LIN {X 0,Y 193.255,Z 819.241,A -85,B 0,C 180,E1 -22296.988,E2 -22296.988} C_VEL
LIN {X 0,Y 197.064,Z 813.143,A -85,B 0,C 180,E1 -22300.279,E2 -22300.279} C_VEL
LIN {X 0,Y 201.414,Z 805.399,A -85,B 0,C 180,E1 -22303.403,E2 -22303.403} C_VEL
LIN {X 0,Y 205.369,Z 797.537,A -85,B 0,C 180,E1 -22305.868,E2 -22305.868} C_VEL
LIN {X 0,Y 209.515,Z 788.24,A -85,B 0,C 180,E1 -22308.163,E2 -22308.163} C_VEL
LIN {X 0,Y 213.305,Z 778.652,A -85,B 0,C 180,E1 -22310.013,E2 -22310.013} C_VEL
LIN {X 0,Y 216.814,Z 768.226,A -85,B 0,C 180,E1 -22311.613,E2 -22311.613} C_VEL
LIN {X 0,Y 219.996,Z 756.796,A -85,B 0,C 180,E1 -22312.978,E2 -22312.978} C_VEL
LIN {X 0,Y 222.629,Z 744.096,A -85,B 0,C 180,E1 -22314.141,E2 -22314.141} C_VEL
LIN {X 0,Y 224.529,Z 731.563,A -85,B 0,C 180,E1 -22314.927,E2 -22314.927} C_VEL
LIN {X 0,Y 227.202,Z 703.845,A -85,B 0,C 180,E1 -22315.948,E2 -22315.948} C_VEL
LIN {X 0,Y 228.654,Z 686.695,A -85,B 0,C 180,E1 -22316.58,E2 -22316.58} C_VEL
LIN {X 0,Y 224.169,Z 676.859,A -85,B 0,C 180,E1 -22318.997,E2 -22318.997} C_VEL
LIN {X 0,Y 221.19,Z 671.533,A -85,B 0,C 180,E1 -22320.701,E2 -22320.701} C_VEL
LIN {X 0,Y 216.957,Z 664.335,A -85,B 0,C 180,E1 -22323.435,E2 -22323.435} C_VEL
LIN {X 0,Y 214.368,Z 660.748,A -85,B 0,C 180,E1 -22325.332,E2 -22325.332} C_VEL
LIN {X 0,Y 211.647,Z 657.239,A -85,B 0,C 180,E1 -22327.574,E2 -22327.574} C_VEL
LIN {X 0,Y 210.827,Z 655.899,A -85,B 0,C 180,E1 -22328.388,E2 -22328.388} C_VEL
LIN {X 0,Y 208.392,Z 652.958,A -85,B 0,C 180,E1 -22330.962,E2 -22330.962} C_VEL
LIN {X 0,Y 207.628,Z 651.927,A -85,B 0,C 180,E1 -22331.967,E2 -22331.967} C_VEL
LIN {X 0,Y 204.394,Z 648.519,A -85,B 0,C 180,E1 -22338.028,E2 -22338.028} C_VEL
LIN {X 0,Y 203.914,Z 648.189,A -85,B 0,C 180,E1 -22340.162,E2 -22340.162} C_VEL
LIN {X 0,Y 203.877,Z 648.812,A -85,B 0,C 180,E1 -22344.436,E2 -22344.436} C_VEL
LIN {X 0,Y 204.528,Z 650.008,A -85,B 0,C 180,E1 -22347.139,E2 -22347.139} C_VEL
LIN {X 0,Y 206.714,Z 654.204,A -85,B 0,C 180,E1 -22351.648,E2 -22351.648} C_VEL
LIN {X 0,Y 209.182,Z 657.668,A -85,B 0,C 180,E1 -22354.733,E2 -22354.733} C_VEL
LIN {X 0,Y 212.852,Z 664.058,A -85,B 0,C 180,E1 -22358.308,E2 -22358.308} C_VEL
LIN {X 0,Y 216.137,Z 670.151,A -85,B 0,C 180,E1 -22360.912,E2 -22360.912} C_VEL
LIN {X 0,Y 219.121,Z 675.87,A -85,B 0,C 180,E1 -22362.932,E2 -22362.932} C_VEL
LIN {X 0,Y 222.15,Z 682.225,A -85,B 0,C 180,E1 -22364.816,E2 -22364.816} C_VEL
LIN {X 0,Y 225.466,Z 690.402,A -85,B 0,C 180,E1 -22366.748,E2 -22366.748} C_VEL
LIN {X 0,Y 227.388,Z 695.915,A -85,B 0,C 180,E1 -22367.832,E2 -22367.832} C_VEL
LIN {X 0,Y 227.649,Z 702.504,A -85,B 0,C 180,E1 -22368.353,E2 -22368.353} C_VEL
LIN {X 0,Y 226.563,Z 715.23,A -85,B 0,C 180,E1 -22368.815,E2 -22368.815} C_VEL
LIN {X 0,Y 225.654,Z 721.062,A -85,B 0,C 180,E1 -22368.881,E2 -22368.881} C_VEL
LIN {X 0,Y 220.375,Z 740.084,A -85,B 0,C 180,E1 -22368.379,E2 -22368.379} C_VEL
LIN {X 0,Y 219.234,Z 745.859,A -85,B 0,C 180,E1 -22368.517,E2 -22368.517} C_VEL
LIN {X 0,Y 216.729,Z 758.978,A -85,B 0,C 180,E1 -22369.31,E2 -22369.31} C_VEL
LIN {X 0,Y 213.46,Z 771.436,A -85,B 0,C 180,E1 -22370.365,E2 -22370.365} C_VEL
LIN {X 0,Y 209.794,Z 782.932,A -85,B 0,C 180,E1 -22371.704,E2 -22371.704} C_VEL
LIN {X 0,Y 205.342,Z 794.569,A -85,B 0,C 180,E1 -22373.512,E2 -22373.512} C_VEL
LIN {X 0,Y 201.089,Z 804.071,A -85,B 0,C 180,E1 -22375.395,E2 -22375.395} C_VEL
LIN {X 0,Y 196.832,Z 812.801,A -85,B 0,C 180,E1 -22377.617,E2 -22377.617} C_VEL
LIN {X 0,Y 192.143,Z 821.48,A -85,B 0,C 180,E1 -22380.411,E2 -22380.411} C_VEL
LIN {X 0,Y 188.053,Z 828.489,A -85,B 0,C 180,E1 -22383.355,E2 -22383.355} C_VEL
LIN {X 0,Y 184.661,Z 834.168,A -85,B 0,C 180,E1 -22386.446,E2 -22386.446} C_VEL
LIN {X 0,Y 181.753,Z 838.705,A -85,B 0,C 180,E1 -22389.635,E2 -22389.635} C_VEL
LIN {X 0,Y 178.675,Z 843.171,A -85,B 0,C 180,E1 -22394.018,E2 -22394.018} C_VEL
LIN {X 0,Y 177.676,Z 844.782,A -85,B 0,C 180,E1 -22396.271,E2 -22396.271} C_VEL
LIN {X 0,Y 176.453,Z 846.754,A -85,B 0,C 180,E1 -22400.833,E2 -22400.833} C_VEL
LIN {X 0,Y 176.148,Z 847.203,A -85,B 0,C 180,E1 -22405.423,E2 -22405.423} C_VEL
LIN {X 0,Y 176.258,Z 846.809,A -85,B 0,C 180,E1 -22407.715,E2 -22407.715} C_VEL
LIN {X 0,Y 176.431,Z 845.994,A -85,B 0,C 180,E1 -22410,E2 -22410} C_VEL
LIN {X 0,Y 176.296,Z 844.734,A -85,B 0,C 180,E1 -22412.285,E2 -22412.285} C_VEL
LIN {X 0,Y 176.257,Z 841.979,A -85,B 0,C 180,E1 -22415.721,E2 -22415.721} C_VEL
LIN {X 0,Y 176.569,Z 838.131,A -85,B 0,C 180,E1 -22419.161,E2 -22419.161} C_VEL
LIN {X 0,Y 177.28,Z 833.082,A -85,B 0,C 180,E1 -22422.594,E2 -22422.594} C_VEL
LIN {X 0,Y 178.531,Z 826.688,A -85,B 0,C 180,E1 -22425.995,E2 -22425.995} C_VEL
LIN {X 0,Y 180.337,Z 818.624,A -85,B 0,C 180,E1 -22429.345,E2 -22429.345} C_VEL
LIN {X 0,Y 182.337,Z 809.868,A -85,B 0,C 180,E1 -22432.239,E2 -22432.239} C_VEL
LIN {X 0,Y 184.548,Z 800.323,A -85,B 0,C 180,E1 -22434.765,E2 -22434.765} C_VEL
LIN {X 0,Y 186.774,Z 790.459,A -85,B 0,C 180,E1 -22436.842,E2 -22436.842} C_VEL
LIN {X 0,Y 189.283,Z 778.076,A -85,B 0,C 180,E1 -22438.86,E2 -22438.86} C_VEL
LIN {X 0,Y 191.275,Z 766.071,A -85,B 0,C 180,E1 -22440.345,E2 -22440.345} C_VEL
LIN {X 0,Y 192.959,Z 753.018,A -85,B 0,C 180,E1 -22441.495,E2 -22441.495} C_VEL
LIN {X 0,Y 194.105,Z 739.399,A -85,B 0,C 180,E1 -22442.279,E2 -22442.279} C_VEL
LIN {X 0,Y 196.335,Z 697.108,A -85,B 0,C 180,E1 -22444.02,E2 -22444.02} C_VEL
LIN {X 0,Y 193.323,Z 669.983,A -85,B 0,C 180,E1 -22445.752,E2 -22445.752} C_VEL
LIN {X 0,Y 184.7,Z 646.505,A -85,B 0,C 180,E1 -22448.296,E2 -22448.296} C_VEL
LIN {X 0,Y 180.166,Z 635.4,A -85,B 0,C 180,E1 -22449.717,E2 -22449.717} C_VEL
LIN {X 0,Y 178.504,Z 628.254,A -85,B 0,C 180,E1 -22453.774,E2 -22453.774} C_VEL
LIN {X 0,Y 178.451,Z 628.257,A -85,B 0,C 180,E1 -22458.44,E2 -22458.44} C_VEL
LIN {X 0,Y 178.489,Z 628.251,A -85,B 0,C 180,E1 -22461.951,E2 -22461.951} C_VEL
LIN {X 0,Y 178.49,Z 628.253,A -85,B 0,C 180,E1 -22466.546,E2 -22466.546} C_VEL
LIN {X 0,Y 178.522,Z 628.245,A -85,B 0,C 180,E1 -22470.005,E2 -22470.005} C_VEL
LIN {X 0,Y 178.518,Z 628.242,A -85,B 0,C 180,E1 -22474.884,E2 -22474.884} C_VEL
LIN {X 0,Y 178.619,Z 628.229,A -85,B 0,C 180,E1 -22480.785,E2 -22480.785} C_VEL
LIN {X 0,Y 178.657,Z 628.231,A -85,B 0,C 180,E1 -22486.347,E2 -22486.347} C_VEL
LIN {X 0,Y 178.934,Z 628.183,A -85,B 0,C 180,E1 -22490.96,E2 -22490.96} C_VEL
LIN {X 0,Y 179.149,Z 628.165,A -85,B 0,C 180,E1 -22497.751,E2 -22497.751} C_VEL
LIN {X 0,Y 179.368,Z 628.128,A -85,B 0,C 180,E1 -22499.999,E2 -22499.999} C_VEL
LIN {X 0,Y 178.87,Z 628.2,A -85,B 0,C 180,E1 -22504.506,E2 -22504.506} C_VEL
LIN {X 0,Y 178.958,Z 628.19,A -85,B 0,C 180,E1 -22509.037,E2 -22509.037} C_VEL
LIN {X 0,Y 178.655,Z 628.211,A -85,B 0,C 180,E1 -22513.651,E2 -22513.651} C_VEL
LIN {X 0,Y 178.618,Z 628.233,A -85,B 0,C 180,E1 -22519.215,E2 -22519.215} C_VEL
LIN {X 0,Y 178.52,Z 628.228,A -85,B 0,C 180,E1 -22525.117,E2 -22525.117} C_VEL
LIN {X 0,Y 178.517,Z 628.244,A -85,B 0,C 180,E1 -22529.992,E2 -22529.992} C_VEL
LIN {X 0,Y 178.479,Z 628.247,A -85,B 0,C 180,E1 -22534.219,E2 -22534.219} C_VEL
LIN {X 0,Y 178.468,Z 628.24,A -85,B 0,C 180,E1 -22539.054,E2 -22539.054} C_VEL
LIN {X 0,Y 178.495,Z 628.247,A -85,B 0,C 180,E1 -22542.015,E2 -22542.015} C_VEL
LIN {X 0,Y 178.512,Z 628.247,A -85,B 0,C 180,E1 -22545.124,E2 -22545.124} C_VEL
LIN {X 0,Y 178.443,Z 628.243,A -85,B 0,C 180,E1 -22548.443,E2 -22548.443} C_VEL
LIN {X 0,Y 178.445,Z 628.255,A -85,B 0,C 180,E1 -22553.789,E2 -22553.789} C_VEL
LIN {X 0,Y 178.485,Z 628.25,A -85,B 0,C 180,E1 -22556.547,E2 -22556.547} C_VEL
LIN {X 0,Y 178.518,Z 628.236,A -85,B 0,C 180,E1 -22560.007,E2 -22560.007} C_VEL
LIN {X 0,Y 178.531,Z 628.245,A -85,B 0,C 180,E1 -22564.876,E2 -22564.876} C_VEL
LIN {X 0,Y 178.635,Z 628.234,A -85,B 0,C 180,E1 -22570.77,E2 -22570.77} C_VEL
LIN {X 0,Y 178.672,Z 628.226,A -85,B 0,C 180,E1 -22574.018,E2 -22574.018} C_VEL
LIN {X 0,Y 178.858,Z 628.201,A -85,B 0,C 180,E1 -22579.21,E2 -22579.21} C_VEL
LIN {X 0,Y 178.922,Z 628.195,A -85,B 0,C 180,E1 -22583.233,E2 -22583.233} C_VEL
LIN {X 0,Y 179.151,Z 628.166,A -85,B 0,C 180,E1 -22587.752,E2 -22587.752} C_VEL
LIN {X 0,Y 179.368,Z 628.139,A -85,B 0,C 180,E1 -22590,E2 -22590} C_VEL
LIN {X 0,Y 178.881,Z 628.202,A -85,B 0,C 180,E1 -22595.637,E2 -22595.637} C_VEL
LIN {X 0,Y 179.948,Z 631.144,A -85,B 0,C 180,E1 -22596.025,E2 -22596.025} C_VEL
LIN {X 0,Y 185.16,Z 641.428,A -85,B 0,C 180,E1 -22597.469,E2 -22597.469} C_VEL
LIN {X 0,Y 194.413,Z 662.027,A -85,B 0,C 180,E1 -22599.952,E2 -22599.952} C_VEL
LIN {X 0,Y 197.42,Z 669.88,A -85,B 0,C 180,E1 -22600.761,E2 -22600.761} C_VEL
LIN {X 0,Y 194.067,Z 726.965,A -85,B 0,C 180,E1 -22603.105,E2 -22603.105} C_VEL
LIN {X 0,Y 192.789,Z 741.069,A -85,B 0,C 180,E1 -22604.114,E2 -22604.114} C_VEL
LIN {X 0,Y 191.209,Z 753.099,A -85,B 0,C 180,E1 -22605.353,E2 -22605.353} C_VEL
LIN {X 0,Y 189.203,Z 765.765,A -85,B 0,C 180,E1 -22607.14,E2 -22607.14} C_VEL
LIN {X 0,Y 186.911,Z 777.168,A -85,B 0,C 180,E1 -22609.208,E2 -22609.208} C_VEL
LIN {X 0,Y 184.516,Z 788.204,A -85,B 0,C 180,E1 -22611.799,E2 -22611.799} C_VEL
LIN {X 0,Y 182.331,Z 797.648,A -85,B 0,C 180,E1 -22614.597,E2 -22614.597} C_VEL
LIN {X 0,Y 180.603,Z 804.839,A -85,B 0,C 180,E1 -22617.225,E2 -22617.225} C_VEL
LIN {X 0,Y 178.814,Z 812.54,A -85,B 0,C 180,E1 -22620.726,E2 -22620.726} C_VEL
LIN {X 0,Y 177.686,Z 817.952,A -85,B 0,C 180,E1 -22623.841,E2 -22623.841} C_VEL
LIN {X 0,Y 176.654,Z 822.661,A -85,B 0,C 180,E1 -22627.283,E2 -22627.283} C_VEL
LIN {X 0,Y 176.052,Z 826.166,A -85,B 0,C 180,E1 -22630.672,E2 -22630.672} C_VEL
LIN {X 0,Y 175.779,Z 828.627,A -85,B 0,C 180,E1 -22633.974,E2 -22633.974} C_VEL
LIN {X 0,Y 175.887,Z 830.168,A -85,B 0,C 180,E1 -22637.214,E2 -22637.214} C_VEL
LIN {X 0,Y 176.397,Z 830.904,A -85,B 0,C 180,E1 -22640.398,E2 -22640.398} C_VEL
LIN {X 0,Y 177.293,Z 830.896,A -85,B 0,C 180,E1 -22643.517,E2 -22643.517} C_VEL
LIN {X 0,Y 178.469,Z 830.163,A -85,B 0,C 180,E1 -22646.544,E2 -22646.544} C_VEL
LIN {X 0,Y 180.914,Z 827.727,A -85,B 0,C 180,E1 -22650.95,E2 -22650.95} C_VEL
LIN {X 0,Y 184.196,Z 823.729,A -85,B 0,C 180,E1 -22655.185,E2 -22655.185} C_VEL
LIN {X 0,Y 186.898,Z 820.049,A -85,B 0,C 180,E1 -22657.913,E2 -22657.913} C_VEL
LIN {X 0,Y 191.103,Z 813.791,A -85,B 0,C 180,E1 -22661.436,E2 -22661.436} C_VEL
LIN {X 0,Y 195.881,Z 805.777,A -85,B 0,C 180,E1 -22664.742,E2 -22664.742} C_VEL
LIN {X 0,Y 200.281,Z 797.617,A -85,B 0,C 180,E1 -22667.333,E2 -22667.333} C_VEL
LIN {X 0,Y 204.6,Z 788.461,A -85,B 0,C 180,E1 -22669.612,E2 -22669.612} C_VEL
LIN {X 0,Y 208.661,Z 778.579,A -85,B 0,C 180,E1 -22671.527,E2 -22671.527} C_VEL
LIN {X 0,Y 212.355,Z 767.997,A -85,B 0,C 180,E1 -22673.141,E2 -22673.141} C_VEL
LIN {X 0,Y 215.884,Z 755.621,A -85,B 0,C 180,E1 -22674.587,E2 -22674.587} C_VEL
LIN {X 0,Y 218.71,Z 741.789,A -85,B 0,C 180,E1 -22675.803,E2 -22675.803} C_VEL
LIN {X 0,Y 220.689,Z 728.831,A -85,B 0,C 180,E1 -22676.528,E2 -22676.528} C_VEL
LIN {X 0,Y 224.387,Z 689.741,A -85,B 0,C 180,E1 -22677.957,E2 -22677.957} C_VEL
LIN {X 0,Y 220.462,Z 680.956,A -85,B 0,C 180,E1 -22680.254,E2 -22680.254} C_VEL
LIN {X 0,Y 217.485,Z 675.634,A -85,B 0,C 180,E1 -22682.135,E2 -22682.135} C_VEL
LIN {X 0,Y 214.316,Z 670.033,A -85,B 0,C 180,E1 -22684.4,E2 -22684.4} C_VEL
LIN {X 0,Y 212.355,Z 667.205,A -85,B 0,C 180,E1 -22685.919,E2 -22685.919} C_VEL
LIN {X 0,Y 209.817,Z 663.776,A -85,B 0,C 180,E1 -22688.155,E2 -22688.155} C_VEL
LIN {X 0,Y 208.904,Z 662.359,A -85,B 0,C 180,E1 -22689.093,E2 -22689.093} C_VEL
LIN {X 0,Y 206.613,Z 659.249,A -85,B 0,C 180,E1 -22691.777,E2 -22691.777} C_VEL
LIN {X 0,Y 204.131,Z 656.773,A -85,B 0,C 180,E1 -22695.732,E2 -22695.732} C_VEL
LIN {X 0,Y 202.982,Z 655.155,A -85,B 0,C 180,E1 -22699.315,E2 -22699.315} C_VEL
LIN {X 0,Y 202.722,Z 655.724,A -85,B 0,C 180,E1 -22704.055,E2 -22704.055} C_VEL
LIN {X 0,Y 203.304,Z 656.974,A -85,B 0,C 180,E1 -22706.858,E2 -22706.858} C_VEL
LIN {X 0,Y 205.332,Z 661.087,A -85,B 0,C 180,E1 -22711.314,E2 -22711.314} C_VEL
LIN {X 0,Y 207.468,Z 664.234,A -85,B 0,C 180,E1 -22714.165,E2 -22714.165} C_VEL
LIN {X 0,Y 210.824,Z 670.507,A -85,B 0,C 180,E1 -22717.679,E2 -22717.679} C_VEL
LIN {X 0,Y 213.784,Z 676.227,A -85,B 0,C 180,E1 -22720.165,E2 -22720.165} C_VEL
LIN {X 0,Y 216.518,Z 681.807,A -85,B 0,C 180,E1 -22722.165,E2 -22722.165} C_VEL
LIN {X 0,Y 219.628,Z 688.985,A -85,B 0,C 180,E1 -22724.268,E2 -22724.268} C_VEL
LIN {X 0,Y 222.785,Z 697.42,A -85,B 0,C 180,E1 -22726.21,E2 -22726.21} C_VEL
LIN {X 0,Y 223.392,Z 699.733,A -85,B 0,C 180,E1 -22726.617,E2 -22726.617} C_VEL
LIN {X 0,Y 223.432,Z 704.022,A -85,B 0,C 180,E1 -22726.941,E2 -22726.941} C_VEL
LIN {X 0,Y 219.671,Z 742.712,A -85,B 0,C 180,E1 -22728.368,E2 -22728.368} C_VEL
LIN {X 0,Y 219.234,Z 745.859,A -85,B 0,C 180,E1 -22728.517,E2 -22728.517} C_VEL
LIN {X 0,Y 217.892,Z 751.602,A -85,B 0,C 180,E1 -22728.671,E2 -22728.671} C_VEL
LIN {X 0,Y 214.123,Z 760.815,A -85,B 0,C 180,E1 -22728.656,E2 -22728.656} C_VEL
LIN {X 0,Y 209.913,Z 769.753,A -85,B 0,C 180,E1 -22728.808,E2 -22728.808} C_VEL
LIN {X 0,Y 207.885,Z 775.051,A -85,B 0,C 180,E1 -22729.235,E2 -22729.235} C_VEL
LIN {X 0,Y 203.861,Z 786.341,A -85,B 0,C 180,E1 -22730.695,E2 -22730.695} C_VEL
LIN {X 0,Y 199.266,Z 797.289,A -85,B 0,C 180,E1 -22732.527,E2 -22732.527} C_VEL
LIN {X 0,Y 194.433,Z 807.146,A -85,B 0,C 180,E1 -22734.667,E2 -22734.667} C_VEL
LIN {X 0,Y 189.214,Z 816.785,A -85,B 0,C 180,E1 -22737.414,E2 -22737.414} C_VEL
LIN {X 0,Y 184.549,Z 824.58,A -85,B 0,C 180,E1 -22740.327,E2 -22740.327} C_VEL
LIN {X 0,Y 180.52,Z 830.911,A -85,B 0,C 180,E1 -22743.405,E2 -22743.405} C_VEL
LIN {X 0,Y 177.047,Z 836.044,A -85,B 0,C 180,E1 -22746.613,E2 -22746.613} C_VEL
LIN {X 0,Y 174.21,Z 840.088,A -85,B 0,C 180,E1 -22749.946,E2 -22749.946} C_VEL
LIN {X 0,Y 171.842,Z 843.142,A -85,B 0,C 180,E1 -22753.365,E2 -22753.365} C_VEL
LIN {X 0,Y 169.976,Z 845.75,A -85,B 0,C 180,E1 -22758.069,E2 -22758.069} C_VEL
LIN {X 0,Y 169.143,Z 846.844,A -85,B 0,C 180,E1 -22762.84,E2 -22762.84} C_VEL
LIN {X 0,Y 169.107,Z 846.677,A -85,B 0,C 180,E1 -22765.905,E2 -22765.905} C_VEL
LIN {X 0,Y 169.368,Z 845.442,A -85,B 0,C 180,E1 -22770,E2 -22770} C_VEL
LIN {X 0,Y 169.218,Z 844.128,A -85,B 0,C 180,E1 -22772.38,E2 -22772.38} C_VEL
LIN {X 0,Y 169.182,Z 841.259,A -85,B 0,C 180,E1 -22775.961,E2 -22775.961} C_VEL
LIN {X 0,Y 169.552,Z 837.296,A -85,B 0,C 180,E1 -22779.544,E2 -22779.544} C_VEL
LIN {X 0,Y 170.491,Z 831.089,A -85,B 0,C 180,E1 -22783.711,E2 -22783.711} C_VEL
LIN {X 0,Y 172.01,Z 824.265,A -85,B 0,C 180,E1 -22787.23,E2 -22787.23} C_VEL
LIN {X 0,Y 173.935,Z 815.717,A -85,B 0,C 180,E1 -22790.704,E2 -22790.704} C_VEL
LIN {X 0,Y 176.122,Z 806.909,A -85,B 0,C 180,E1 -22793.518,E2 -22793.518} C_VEL
LIN {X 0,Y 178.694,Z 796.079,A -85,B 0,C 180,E1 -22796.26,E2 -22796.26} C_VEL
LIN {X 0,Y 181.047,Z 785.315,A -85,B 0,C 180,E1 -22798.393,E2 -22798.393} C_VEL
LIN {X 0,Y 183.375,Z 773.376,A -85,B 0,C 180,E1 -22800.2,E2 -22800.2} C_VEL
LIN {X 0,Y 185.339,Z 761.168,A -85,B 0,C 180,E1 -22801.584,E2 -22801.584} C_VEL
LIN {X 0,Y 186.888,Z 747.853,A -85,B 0,C 180,E1 -22802.642,E2 -22802.642} C_VEL
LIN {X 0,Y 188.123,Z 729.575,A -85,B 0,C 180,E1 -22803.517,E2 -22803.517} C_VEL
LIN {X 0,Y 189.825,Z 697.425,A -85,B 0,C 180,E1 -22804.888,E2 -22804.888} C_VEL
LIN {X 0,Y 187.03,Z 672.005,A -85,B 0,C 180,E1 -22806.593,E2 -22806.593} C_VEL
LIN {X 0,Y 178.857,Z 649.667,A -85,B 0,C 180,E1 -22809.106,E2 -22809.106} C_VEL
LIN {X 0,Y 172.86,Z 635.106,A -85,B 0,C 180,E1 -22811.043,E2 -22811.043} C_VEL
LIN {X 0,Y 171.42,Z 629.135,A -85,B 0,C 180,E1 -22814.657,E2 -22814.657} C_VEL
LIN {X 0,Y 171.383,Z 629.136,A -85,B 0,C 180,E1 -22818.994,E2 -22818.994} C_VEL
LIN {X 0,Y 171.436,Z 629.13,A -85,B 0,C 180,E1 -22822.052,E2 -22822.052} C_VEL
LIN {X 0,Y 171.419,Z 629.132,A -85,B 0,C 180,E1 -22827.791,E2 -22827.791} C_VEL
LIN {X 0,Y 171.448,Z 629.127,A -85,B 0,C 180,E1 -22830.533,E2 -22830.533} C_VEL
LIN {X 0,Y 171.443,Z 629.128,A -85,B 0,C 180,E1 -22835.798,E2 -22835.798} C_VEL
LIN {X 0,Y 171.575,Z 629.106,A -85,B 0,C 180,E1 -22840.87,E2 -22840.87} C_VEL
LIN {X 0,Y 171.574,Z 629.114,A -85,B 0,C 180,E1 -22845.771,E2 -22845.771} C_VEL
LIN {X 0,Y 171.869,Z 629.062,A -85,B 0,C 180,E1 -22850.585,E2 -22850.585} C_VEL
LIN {X 0,Y 171.818,Z 629.084,A -85,B 0,C 180,E1 -22855.306,E2 -22855.306} C_VEL
LIN {X 0,Y 172.33,Z 629.004,A -85,B 0,C 180,E1 -22859.999,E2 -22859.999} C_VEL
LIN {X 0,Y 171.819,Z 629.078,A -85,B 0,C 180,E1 -22864.691,E2 -22864.691} C_VEL
LIN {X 0,Y 171.886,Z 629.07,A -85,B 0,C 180,E1 -22869.412,E2 -22869.412} C_VEL
LIN {X 0,Y 171.572,Z 629.096,A -85,B 0,C 180,E1 -22874.226,E2 -22874.226} C_VEL
LIN {X 0,Y 171.54,Z 629.116,A -85,B 0,C 180,E1 -22879.561,E2 -22879.561} C_VEL
LIN {X 0,Y 171.457,Z 629.106,A -85,B 0,C 180,E1 -22885.61,E2 -22885.61} C_VEL
LIN {X 0,Y 171.435,Z 629.128,A -85,B 0,C 180,E1 -22890.585,E2 -22890.585} C_VEL
LIN {X 0,Y 171.399,Z 629.127,A -85,B 0,C 180,E1 -22895.032,E2 -22895.032} C_VEL
LIN {X 0,Y 171.422,Z 629.115,A -85,B 0,C 180,E1 -22898.836,E2 -22898.836} C_VEL
LIN {X 0,Y 171.437,Z 629.131,A -85,B 0,C 180,E1 -22904.178,E2 -22904.178} C_VEL
LIN {X 0,Y 171.368,Z 629.122,A -85,B 0,C 180,E1 -22908.992,E2 -22908.992} C_VEL
LIN {X 0,Y 171.413,Z 629.126,A -85,B 0,C 180,E1 -22912.049,E2 -22912.049} C_VEL
LIN {X 0,Y 171.406,Z 629.133,A -85,B 0,C 180,E1 -22915.087,E2 -22915.087} C_VEL
LIN {X 0,Y 171.444,Z 629.119,A -85,B 0,C 180,E1 -22920.534,E2 -22920.534} C_VEL
LIN {X 0,Y 171.455,Z 629.124,A -85,B 0,C 180,E1 -22925.802,E2 -22925.802} C_VEL
LIN {X 0,Y 171.592,Z 629.111,A -85,B 0,C 180,E1 -22930.874,E2 -22930.874} C_VEL
LIN {X 0,Y 171.61,Z 629.104,A -85,B 0,C 180,E1 -22935.776,E2 -22935.776} C_VEL
LIN {X 0,Y 171.886,Z 629.071,A -85,B 0,C 180,E1 -22940.587,E2 -22940.587} C_VEL
LIN {X 0,Y 171.82,Z 629.079,A -85,B 0,C 180,E1 -22945.308,E2 -22945.308} C_VEL
LIN {X 0,Y 172.331,Z 629.015,A -85,B 0,C 180,E1 -22950,E2 -22950} C_VEL
LIN {X 0,Y 171.853,Z 629.187,A -85,B 0,C 180,E1 -22954.398,E2 -22954.398} C_VEL
LIN {X 0,Y 172.916,Z 632.075,A -85,B 0,C 180,E1 -22954.772,E2 -22954.772} C_VEL
LIN {X 0,Y 179.165,Z 644.151,A -85,B 0,C 180,E1 -22956.602,E2 -22956.602} C_VEL
LIN {X 0,Y 188.576,Z 665.333,A -85,B 0,C 180,E1 -22959.243,E2 -22959.243} C_VEL
LIN {X 0,Y 190.943,Z 671.332,A -85,B 0,C 180,E1 -22959.905,E2 -22959.905} C_VEL
LIN {X 0,Y 187.502,Z 728.004,A -85,B 0,C 180,E1 -22962.32,E2 -22962.32} C_VEL
LIN {X 0,Y 186.123,Z 742.074,A -85,B 0,C 180,E1 -22963.372,E2 -22963.372} C_VEL
LIN {X 0,Y 184.376,Z 754.774,A -85,B 0,C 180,E1 -22964.768,E2 -22964.768} C_VEL
LIN {X 0,Y 182.165,Z 767.808,A -85,B 0,C 180,E1 -22966.717,E2 -22966.717} C_VEL
LIN {X 0,Y 179.794,Z 778.928,A -85,B 0,C 180,E1 -22968.883,E2 -22968.883} C_VEL
LIN {X 0,Y 177.458,Z 789.373,A -85,B 0,C 180,E1 -22971.489,E2 -22971.489} C_VEL
LIN {X 0,Y 175.287,Z 798.294,A -85,B 0,C 180,E1 -22974.265,E2 -22974.265} C_VEL
LIN {X 0,Y 173.252,Z 806.498,A -85,B 0,C 180,E1 -22977.451,E2 -22977.451} C_VEL
LIN {X 0,Y 171.377,Z 814.444,A -85,B 0,C 180,E1 -22981.416,E2 -22981.416} C_VEL
LIN {X 0,Y 170.085,Z 820.498,A -85,B 0,C 180,E1 -22985.343,E2 -22985.343} C_VEL
LIN {X 0,Y 169.32,Z 824.241,A -85,B 0,C 180,E1 -22988.506,E2 -22988.506} C_VEL
LIN {X 0,Y 168.818,Z 827.197,A -85,B 0,C 180,E1 -22991.765,E2 -22991.765} C_VEL
LIN {X 0,Y 168.67,Z 829.377,A -85,B 0,C 180,E1 -22995.099,E2 -22995.099} C_VEL
LIN {X 0,Y 168.952,Z 830.775,A -85,B 0,C 180,E1 -22998.481,E2 -22998.481} C_VEL
LIN {X 0,Y 169.674,Z 831.367,A -85,B 0,C 180,E1 -23001.903,E2 -23001.903} C_VEL
LIN {X 0,Y 170.82,Z 831.101,A -85,B 0,C 180,E1 -23005.369,E2 -23005.369} C_VEL
LIN {X 0,Y 172.458,Z 829.969,A -85,B 0,C 180,E1 -23008.845,E2 -23008.845} C_VEL
LIN {X 0,Y 174.623,Z 827.915,A -85,B 0,C 180,E1 -23012.301,E2 -23012.301} C_VEL
LIN {X 0,Y 178.4,Z 823.64,A -85,B 0,C 180,E1 -23016.801,E2 -23016.801} C_VEL
LIN {X 0,Y 182.127,Z 818.782,A -85,B 0,C 180,E1 -23020.268,E2 -23020.268} C_VEL
LIN {X 0,Y 186.531,Z 812.524,A -85,B 0,C 180,E1 -23023.587,E2 -23023.587} C_VEL
LIN {X 0,Y 190.671,Z 805.932,A -85,B 0,C 180,E1 -23026.282,E2 -23026.282} C_VEL
LIN {X 0,Y 195.402,Z 797.602,A -85,B 0,C 180,E1 -23028.931,E2 -23028.931} C_VEL
LIN {X 0,Y 199.788,Z 788.657,A -85,B 0,C 180,E1 -23031.159,E2 -23031.159} C_VEL
LIN {X 0,Y 204.715,Z 777.254,A -85,B 0,C 180,E1 -23033.321,E2 -23033.321} C_VEL
LIN {X 0,Y 208.606,Z 766.378,A -85,B 0,C 180,E1 -23034.928,E2 -23034.928} C_VEL
LIN {X 0,Y 212.098,Z 754.066,A -85,B 0,C 180,E1 -23036.313,E2 -23036.313} C_VEL
LIN {X 0,Y 214.799,Z 741.328,A -85,B 0,C 180,E1 -23037.389,E2 -23037.389} C_VEL
LIN {X 0,Y 216.842,Z 727.728,A -85,B 0,C 180,E1 -23038.116,E2 -23038.116} C_VEL
LIN {X 0,Y 220.266,Z 692.867,A -85,B 0,C 180,E1 -23039.392,E2 -23039.392} C_VEL
LIN {X 0,Y 217.332,Z 686.016,A -85,B 0,C 180,E1 -23041.296,E2 -23041.296} C_VEL
LIN {X 0,Y 212.455,Z 676.772,A -85,B 0,C 180,E1 -23044.82,E2 -23044.82} C_VEL
LIN {X 0,Y 210.296,Z 673.629,A -85,B 0,C 180,E1 -23046.56,E2 -23046.56} C_VEL
LIN {X 0,Y 207.724,Z 669.748,A -85,B 0,C 180,E1 -23049.063,E2 -23049.063} C_VEL
LIN {X 0,Y 204.852,Z 665.669,A -85,B 0,C 180,E1 -23052.615,E2 -23052.615} C_VEL
LIN {X 0,Y 202.178,Z 662.711,A -85,B 0,C 180,E1 -23057.908,E2 -23057.908} C_VEL
LIN {X 0,Y 201.952,Z 662.225,A -85,B 0,C 180,E1 -23058.945,E2 -23058.945} C_VEL
LIN {X 0,Y 201.589,Z 662.693,A -85,B 0,C 180,E1 -23063.831,E2 -23063.831} C_VEL
LIN {X 0,Y 202.065,Z 663.834,A -85,B 0,C 180,E1 -23066.486,E2 -23066.486} C_VEL
LIN {X 0,Y 203.897,Z 667.876,A -85,B 0,C 180,E1 -23070.879,E2 -23070.879} C_VEL
LIN {X 0,Y 205.708,Z 670.713,A -85,B 0,C 180,E1 -23073.505,E2 -23073.505} C_VEL
LIN {X 0,Y 208.728,Z 676.703,A -85,B 0,C 180,E1 -23076.918,E2 -23076.918} C_VEL
LIN {X 0,Y 211.489,Z 682.392,A -85,B 0,C 180,E1 -23079.417,E2 -23079.417} C_VEL
LIN {X 0,Y 213.709,Z 687.227,A -85,B 0,C 180,E1 -23081.204,E2 -23081.204} C_VEL
LIN {X 0,Y 216.981,Z 695.272,A -85,B 0,C 180,E1 -23083.565,E2 -23083.565} C_VEL
LIN {X 0,Y 219.464,Z 702.678,A -85,B 0,C 180,E1 -23085.258,E2 -23085.258} C_VEL
LIN {X 0,Y 219.371,Z 706.135,A -85,B 0,C 180,E1 -23085.483,E2 -23085.483} C_VEL
LIN {X 0,Y 215.645,Z 742.372,A -85,B 0,C 180,E1 -23086.813,E2 -23086.813} C_VEL
LIN {X 0,Y 213.314,Z 755.229,A -85,B 0,C 180,E1 -23087.515,E2 -23087.515} C_VEL
LIN {X 0,Y 210.455,Z 766.797,A -85,B 0,C 180,E1 -23088.418,E2 -23088.418} C_VEL
LIN {X 0,Y 207.885,Z 775.051,A -85,B 0,C 180,E1 -23089.235,E2 -23089.235} C_VEL
LIN {X 0,Y 205.752,Z 780.293,A -85,B 0,C 180,E1 -23089.732,E2 -23089.732} C_VEL
LIN {X 0,Y 200.78,Z 788.644,A -85,B 0,C 180,E1 -23090.271,E2 -23090.271} C_VEL
LIN {X 0,Y 195.395,Z 796.585,A -85,B 0,C 180,E1 -23090.973,E2 -23090.973} C_VEL
LIN {X 0,Y 192.647,Z 801.11,A -85,B 0,C 180,E1 -23091.735,E2 -23091.735} C_VEL
LIN {X 0,Y 187.805,Z 810.021,A -85,B 0,C 180,E1 -23093.887,E2 -23093.887} C_VEL
LIN {X 0,Y 182.508,Z 818.989,A -85,B 0,C 180,E1 -23096.72,E2 -23096.72} C_VEL
LIN {X 0,Y 177.691,Z 826.315,A -85,B 0,C 180,E1 -23099.717,E2 -23099.717} C_VEL
LIN {X 0,Y 172.947,Z 833.114,A -85,B 0,C 180,E1 -23103.449,E2 -23103.449} C_VEL
LIN {X 0,Y 169.449,Z 837.692,A -85,B 0,C 180,E1 -23106.796,E2 -23106.796} C_VEL
LIN {X 0,Y 166.637,Z 841.26,A -85,B 0,C 180,E1 -23110.282,E2 -23110.282} C_VEL
LIN {X 0,Y 163.826,Z 844.505,A -85,B 0,C 180,E1 -23115.085,E2 -23115.085} C_VEL
LIN {X 0,Y 162.388,Z 846.221,A -85,B 0,C 180,E1 -23120.031,E2 -23120.031} C_VEL
LIN {X 0,Y 161.995,Z 846.336,A -85,B 0,C 180,E1 -23125.022,E2 -23125.022} C_VEL
LIN {X 0,Y 162.101,Z 845.81,A -85,B 0,C 180,E1 -23127.515,E2 -23127.515} C_VEL
LIN {X 0,Y 162.304,Z 844.886,A -85,B 0,C 180,E1 -23130,E2 -23130} C_VEL
LIN {X 0,Y 162.128,Z 842.059,A -85,B 0,C 180,E1 -23134.415,E2 -23134.415} C_VEL
LIN {X 0,Y 162.357,Z 837.855,A -85,B 0,C 180,E1 -23138.714,E2 -23138.714} C_VEL
LIN {X 0,Y 163.03,Z 832.934,A -85,B 0,C 180,E1 -23142.447,E2 -23142.447} C_VEL
LIN {X 0,Y 164.288,Z 826.682,A -85,B 0,C 180,E1 -23146.144,E2 -23146.144} C_VEL
LIN {X 0,Y 166.144,Z 818.844,A -85,B 0,C 180,E1 -23149.779,E2 -23149.779} C_VEL
LIN {X 0,Y 168.439,Z 809.552,A -85,B 0,C 180,E1 -23153.145,E2 -23153.145} C_VEL
LIN {X 0,Y 170.86,Z 799.887,A -85,B 0,C 180,E1 -23155.914,E2 -23155.914} C_VEL
LIN {X 0,Y 173.199,Z 790.096,A -85,B 0,C 180,E1 -23158.145,E2 -23158.145} C_VEL
LIN {X 0,Y 175.889,Z 777.837,A -85,B 0,C 180,E1 -23160.294,E2 -23160.294} C_VEL
LIN {X 0,Y 178.168,Z 764.838,A -85,B 0,C 180,E1 -23162.008,E2 -23162.008} C_VEL
LIN {X 0,Y 179.96,Z 751.579,A -85,B 0,C 180,E1 -23163.227,E2 -23163.227} C_VEL
LIN {X 0,Y 181.074,Z 738.919,A -85,B 0,C 180,E1 -23163.996,E2 -23163.996} C_VEL
LIN {X 0,Y 183.407,Z 698.973,A -85,B 0,C 180,E1 -23165.748,E2 -23165.748} C_VEL
LIN {X 0,Y 180.871,Z 674.427,A -85,B 0,C 180,E1 -23167.425,E2 -23167.425} C_VEL
LIN {X 0,Y 173.312,Z 653.402,A -85,B 0,C 180,E1 -23169.884,E2 -23169.884} C_VEL
LIN {X 0,Y 166.716,Z 637.842,A -85,B 0,C 180,E1 -23172.073,E2 -23172.073} C_VEL
LIN {X 0,Y 165.428,Z 634.651,A -85,B 0,C 180,E1 -23172.589,E2 -23172.589} C_VEL
LIN {X 0,Y 164.335,Z 630.018,A -85,B 0,C 180,E1 -23175.549,E2 -23175.549} C_VEL
LIN {X 0,Y 164.345,Z 630.015,A -85,B 0,C 180,E1 -23180.33,E2 -23180.33} C_VEL
LIN {X 0,Y 164.344,Z 630.014,A -85,B 0,C 180,E1 -23184.34,E2 -23184.34} C_VEL
LIN {X 0,Y 164.39,Z 630.004,A -85,B 0,C 180,E1 -23189.133,E2 -23189.133} C_VEL
LIN {X 0,Y 164.405,Z 629.999,A -85,B 0,C 180,E1 -23194.691,E2 -23194.691} C_VEL
LIN {X 0,Y 164.482,Z 629.993,A -85,B 0,C 180,E1 -23200.05,E2 -23200.05} C_VEL
LIN {X 0,Y 164.522,Z 629.994,A -85,B 0,C 180,E1 -23205.148,E2 -23205.148} C_VEL
LIN {X 0,Y 164.794,Z 629.943,A -85,B 0,C 180,E1 -23210.177,E2 -23210.177} C_VEL
LIN {X 0,Y 164.842,Z 629.945,A -85,B 0,C 180,E1 -23212.65,E2 -23212.65} C_VEL
LIN {X 0,Y 165.046,Z 629.922,A -85,B 0,C 180,E1 -23217.558,E2 -23217.558} C_VEL
LIN {X 0,Y 165.293,Z 629.88,A -85,B 0,C 180,E1 -23219.999,E2 -23219.999} C_VEL
LIN {X 0,Y 164.826,Z 629.951,A -85,B 0,C 180,E1 -23227.085,E2 -23227.085} C_VEL
LIN {X 0,Y 164.738,Z 629.951,A -85,B 0,C 180,E1 -23231.13,E2 -23231.13} C_VEL
LIN {X 0,Y 164.478,Z 629.991,A -85,B 0,C 180,E1 -23237.402,E2 -23237.402} C_VEL
LIN {X 0,Y 164.469,Z 629.995,A -85,B 0,C 180,E1 -23239.988,E2 -23239.988} C_VEL
LIN {X 0,Y 164.383,Z 629.987,A -85,B 0,C 180,E1 -23246.129,E2 -23246.129} C_VEL
LIN {X 0,Y 164.369,Z 630.007,A -85,B 0,C 180,E1 -23251.226,E2 -23251.226} C_VEL
LIN {X 0,Y 164.343,Z 629.996,A -85,B 0,C 180,E1 -23256.775,E2 -23256.775} C_VEL
LIN {X 0,Y 164.364,Z 629.998,A -85,B 0,C 180,E1 -23259.893,E2 -23259.893} C_VEL
LIN {X 0,Y 164.374,Z 630.008,A -85,B 0,C 180,E1 -23263.378,E2 -23263.378} C_VEL
LIN {X 0,Y 164.353,Z 630.006,A -85,B 0,C 180,E1 -23266.83,E2 -23266.83} C_VEL
LIN {X 0,Y 164.31,Z 630.002,A -85,B 0,C 180,E1 -23270.344,E2 -23270.344} C_VEL
LIN {X 0,Y 164.339,Z 630.015,A -85,B 0,C 180,E1 -23274.342,E2 -23274.342} C_VEL
LIN {X 0,Y 164.385,Z 629.995,A -85,B 0,C 180,E1 -23279.134,E2 -23279.134} C_VEL
LIN {X 0,Y 164.413,Z 630.004,A -85,B 0,C 180,E1 -23284.694,E2 -23284.694} C_VEL
LIN {X 0,Y 164.483,Z 629.994,A -85,B 0,C 180,E1 -23290.05,E2 -23290.05} C_VEL
LIN {X 0,Y 164.555,Z 629.984,A -85,B 0,C 180,E1 -23295.152,E2 -23295.152} C_VEL
LIN {X 0,Y 164.806,Z 629.951,A -85,B 0,C 180,E1 -23300.179,E2 -23300.179} C_VEL
LIN {X 0,Y 164.848,Z 629.946,A -85,B 0,C 180,E1 -23302.652,E2 -23302.652} C_VEL
LIN {X 0,Y 165.047,Z 629.922,A -85,B 0,C 180,E1 -23307.56,E2 -23307.56} C_VEL
LIN {X 0,Y 165.293,Z 629.892,A -85,B 0,C 180,E1 -23310,E2 -23310} C_VEL
LIN {X 0,Y 164.945,Z 629.993,A -85,B 0,C 180,E1 -23313.054,E2 -23313.054} C_VEL
LIN {X 0,Y 165.984,Z 632.903,A -85,B 0,C 180,E1 -23313.448,E2 -23313.448} C_VEL
LIN {X 0,Y 173.623,Z 647.842,A -85,B 0,C 180,E1 -23315.808,E2 -23315.808} C_VEL
LIN {X 0,Y 183.294,Z 669.924,A -85,B 0,C 180,E1 -23318.669,E2 -23318.669} C_VEL
LIN {X 0,Y 184.418,Z 672.622,A -85,B 0,C 180,E1 -23318.984,E2 -23318.984} C_VEL
LIN {X 0,Y 180.979,Z 728.277,A -85,B 0,C 180,E1 -23321.453,E2 -23321.453} C_VEL
LIN {X 0,Y 179.571,Z 742.336,A -85,B 0,C 180,E1 -23322.54,E2 -23322.54} C_VEL
LIN {X 0,Y 177.7,Z 755.331,A -85,B 0,C 180,E1 -23324.019,E2 -23324.019} C_VEL
LIN {X 0,Y 175.457,Z 768.059,A -85,B 0,C 180,E1 -23325.991,E2 -23325.991} C_VEL
LIN {X 0,Y 172.876,Z 779.755,A -85,B 0,C 180,E1 -23328.364,E2 -23328.364} C_VEL
LIN {X 0,Y 170.302,Z 790.813,A -85,B 0,C 180,E1 -23331.267,E2 -23331.267} C_VEL
LIN {X 0,Y 168.159,Z 799.255,A -85,B 0,C 180,E1 -23334.05,E2 -23334.05} C_VEL
LIN {X 0,Y 166.101,Z 807.201,A -85,B 0,C 180,E1 -23337.312,E2 -23337.312} C_VEL
LIN {X 0,Y 164.31,Z 814.655,A -85,B 0,C 180,E1 -23341.193,E2 -23341.193} C_VEL
LIN {X 0,Y 163.045,Z 820.387,A -85,B 0,C 180,E1 -23345.019,E2 -23345.019} C_VEL
LIN {X 0,Y 162.166,Z 824.666,A -85,B 0,C 180,E1 -23348.733,E2 -23348.733} C_VEL
LIN {X 0,Y 161.678,Z 827.777,A -85,B 0,C 180,E1 -23352.358,E2 -23352.358} C_VEL
LIN {X 0,Y 161.616,Z 829.916,A -85,B 0,C 180,E1 -23355.913,E2 -23355.913} C_VEL
LIN {X 0,Y 162.37,Z 831.581,A -85,B 0,C 180,E1 -23361.177,E2 -23361.177} C_VEL
LIN {X 0,Y 164.001,Z 831.501,A -85,B 0,C 180,E1 -23366.146,E2 -23366.146} C_VEL
LIN {X 0,Y 165.559,Z 830.573,A -85,B 0,C 180,E1 -23369.378,E2 -23369.378} C_VEL
LIN {X 0,Y 168.689,Z 827.882,A -85,B 0,C 180,E1 -23374.061,E2 -23374.061} C_VEL
LIN {X 0,Y 172.778,Z 823.548,A -85,B 0,C 180,E1 -23378.527,E2 -23378.527} C_VEL
LIN {X 0,Y 177.1,Z 818.28,A -85,B 0,C 180,E1 -23382.248,E2 -23382.248} C_VEL
LIN {X 0,Y 181.578,Z 812.27,A -85,B 0,C 180,E1 -23385.376,E2 -23385.376} C_VEL
LIN {X 0,Y 186.538,Z 804.686,A -85,B 0,C 180,E1 -23388.393,E2 -23388.393} C_VEL
LIN {X 0,Y 191.989,Z 795.253,A -85,B 0,C 180,E1 -23391.243,E2 -23391.243} C_VEL
LIN {X 0,Y 196.456,Z 786.369,A -85,B 0,C 180,E1 -23393.324,E2 -23393.324} C_VEL
LIN {X 0,Y 201.113,Z 775.721,A -85,B 0,C 180,E1 -23395.24,E2 -23395.24} C_VEL
LIN {X 0,Y 205.45,Z 763.54,A -85,B 0,C 180,E1 -23396.92,E2 -23396.92} C_VEL
LIN {X 0,Y 208.927,Z 751.048,A -85,B 0,C 180,E1 -23398.22,E2 -23398.22} C_VEL
LIN {X 0,Y 211.331,Z 739.389,A -85,B 0,C 180,E1 -23399.124,E2 -23399.124} C_VEL
LIN {X 0,Y 213.296,Z 726.116,A -85,B 0,C 180,E1 -23399.782,E2 -23399.782} C_VEL
LIN {X 0,Y 216.366,Z 695.997,A -85,B 0,C 180,E1 -23400.901,E2 -23400.901} C_VEL
LIN {X 0,Y 213.743,Z 689.917,A -85,B 0,C 180,E1 -23402.756,E2 -23402.756} C_VEL
LIN {X 0,Y 209.85,Z 682.389,A -85,B 0,C 180,E1 -23405.858,E2 -23405.858} C_VEL
LIN {X 0,Y 208.313,Z 680.051,A -85,B 0,C 180,E1 -23407.205,E2 -23407.205} C_VEL
LIN {X 0,Y 205.867,Z 676.12,A -85,B 0,C 180,E1 -23409.751,E2 -23409.751} C_VEL
LIN {X 0,Y 203.221,Z 672.293,A -85,B 0,C 180,E1 -23413.312,E2 -23413.312} C_VEL
LIN {X 0,Y 200.811,Z 669.215,A -85,B 0,C 180,E1 -23419.104,E2 -23419.104} C_VEL
LIN {X 0,Y 200.496,Z 669.76,A -85,B 0,C 180,E1 -23423.969,E2 -23423.969} C_VEL
LIN {X 0,Y 200.905,Z 670.913,A -85,B 0,C 180,E1 -23426.38,E2 -23426.38} C_VEL
LIN {X 0,Y 202.705,Z 675.037,A -85,B 0,C 180,E1 -23430.825,E2 -23430.825} C_VEL
LIN {X 0,Y 204.093,Z 677.416,A -85,B 0,C 180,E1 -23432.946,E2 -23432.946} C_VEL
LIN {X 0,Y 206.686,Z 682.846,A -85,B 0,C 180,E1 -23436.125,E2 -23436.125} C_VEL
LIN {X 0,Y 209.135,Z 688.317,A -85,B 0,C 180,E1 -23438.565,E2 -23438.565} C_VEL
LIN {X 0,Y 211.718,Z 694.371,A -85,B 0,C 180,E1 -23440.799,E2 -23440.799} C_VEL
LIN {X 0,Y 214.861,Z 703.03,A -85,B 0,C 180,E1 -23443.212,E2 -23443.212} C_VEL
LIN {X 0,Y 215.701,Z 706.098,A -85,B 0,C 180,E1 -23443.878,E2 -23443.878} C_VEL
LIN {X 0,Y 211.73,Z 742.375,A -85,B 0,C 180,E1 -23445.211,E2 -23445.211} C_VEL
LIN {X 0,Y 209.16,Z 755.914,A -85,B 0,C 180,E1 -23445.965,E2 -23445.965} C_VEL
LIN {X 0,Y 205.909,Z 768.164,A -85,B 0,C 180,E1 -23446.952,E2 -23446.952} C_VEL
LIN {X 0,Y 201.832,Z 780.107,A -85,B 0,C 180,E1 -23448.246,E2 -23448.246} C_VEL
LIN {X 0,Y 197.445,Z 790.961,A -85,B 0,C 180,E1 -23449.824,E2 -23449.824} C_VEL
LIN {X 0,Y 192.647,Z 801.11,A -85,B 0,C 180,E1 -23451.735,E2 -23451.735} C_VEL
LIN {X 0,Y 189.845,Z 805.555,A -85,B 0,C 180,E1 -23452.588,E2 -23452.588} C_VEL
LIN {X 0,Y 181.42,Z 815.094,A -85,B 0,C 180,E1 -23454.318,E2 -23454.318} C_VEL
LIN {X 0,Y 176.838,Z 820.008,A -85,B 0,C 180,E1 -23455.608,E2 -23455.608} C_VEL
LIN {X 0,Y 175.028,Z 822.259,A -85,B 0,C 180,E1 -23456.444,E2 -23456.444} C_VEL
LIN {X 0,Y 170.096,Z 828.942,A -85,B 0,C 180,E1 -23459.593,E2 -23459.593} C_VEL
LIN {X 0,Y 165.825,Z 834.528,A -85,B 0,C 180,E1 -23463.095,E2 -23463.095} C_VEL
LIN {X 0,Y 161.865,Z 839.146,A -85,B 0,C 180,E1 -23466.998,E2 -23466.998} C_VEL
LIN {X 0,Y 158.266,Z 843.021,A -85,B 0,C 180,E1 -23471.89,E2 -23471.89} C_VEL
LIN {X 0,Y 156.015,Z 845.351,A -85,B 0,C 180,E1 -23476.984,E2 -23476.984} C_VEL
LIN {X 0,Y 155.01,Z 846.085,A -85,B 0,C 180,E1 -23482.183,E2 -23482.183} C_VEL
LIN {X 0,Y 155.035,Z 845.305,A -85,B 0,C 180,E1 -23487.402,E2 -23487.402} C_VEL
LIN {X 0,Y 155.241,Z 844.296,A -85,B 0,C 180,E1 -23490,E2 -23490} C_VEL
LIN {X 0,Y 155.067,Z 841.526,A -85,B 0,C 180,E1 -23494.356,E2 -23494.356} C_VEL
LIN {X 0,Y 155.331,Z 836.971,A -85,B 0,C 180,E1 -23499.111,E2 -23499.111} C_VEL
LIN {X 0,Y 156.089,Z 831.905,A -85,B 0,C 180,E1 -23503.01,E2 -23503.01} C_VEL
LIN {X 0,Y 157.467,Z 825.48,A -85,B 0,C 180,E1 -23506.864,E2 -23506.864} C_VEL
LIN {X 0,Y 159.429,Z 817.371,A -85,B 0,C 180,E1 -23510.649,E2 -23510.649} C_VEL
LIN {X 0,Y 161.732,Z 808.597,A -85,B 0,C 180,E1 -23513.889,E2 -23513.889} C_VEL
LIN {X 0,Y 164.175,Z 799.003,A -85,B 0,C 180,E1 -23516.71,E2 -23516.71} C_VEL
LIN {X 0,Y 166.626,Z 789.06,A -85,B 0,C 180,E1 -23519.015,E2 -23519.015} C_VEL
LIN {X 0,Y 169.399,Z 776.623,A -85,B 0,C 180,E1 -23521.237,E2 -23521.237} C_VEL
LIN {X 0,Y 171.582,Z 764.499,A -85,B 0,C 180,E1 -23522.868,E2 -23522.868} C_VEL
LIN {X 0,Y 173.429,Z 751.245,A -85,B 0,C 180,E1 -23524.124,E2 -23524.124} C_VEL
LIN {X 0,Y 174.687,Z 737.639,A -85,B 0,C 180,E1 -23524.96,E2 -23524.96} C_VEL
LIN {X 0,Y 176.921,Z 698.503,A -85,B 0,C 180,E1 -23526.75,E2 -23526.75} C_VEL
LIN {X 0,Y 174.589,Z 676.386,A -85,B 0,C 180,E1 -23528.351,E2 -23528.351} C_VEL
LIN {X 0,Y 166.838,Z 654.722,A -85,B 0,C 180,E1 -23531.034,E2 -23531.034} C_VEL
LIN {X 0,Y 160.792,Z 640.573,A -85,B 0,C 180,E1 -23533.137,E2 -23533.137} C_VEL
LIN {X 0,Y 158.137,Z 634.333,A -85,B 0,C 180,E1 -23534.164,E2 -23534.164} C_VEL
LIN {X 0,Y 157.286,Z 630.894,A -85,B 0,C 180,E1 -23536.459,E2 -23536.459} C_VEL
LIN {X 0,Y 157.271,Z 630.894,A -85,B 0,C 180,E1 -23541.271,E2 -23541.271} C_VEL
LIN {X 0,Y 157.291,Z 630.892,A -85,B 0,C 180,E1 -23544.488,E2 -23544.488} C_VEL
LIN {X 0,Y 157.294,Z 630.891,A -85,B 0,C 180,E1 -23548.094,E2 -23548.094} C_VEL
LIN {X 0,Y 157.314,Z 630.883,A -85,B 0,C 180,E1 -23553.463,E2 -23553.463} C_VEL
LIN {X 0,Y 157.39,Z 630.877,A -85,B 0,C 180,E1 -23559.668,E2 -23559.668} C_VEL
LIN {X 0,Y 157.451,Z 630.872,A -85,B 0,C 180,E1 -23564.464,E2 -23564.464} C_VEL
LIN {X 0,Y 157.722,Z 630.825,A -85,B 0,C 180,E1 -23569.732,E2 -23569.732} C_VEL
LIN {X 0,Y 157.8,Z 630.822,A -85,B 0,C 180,E1 -23572.32,E2 -23572.32} C_VEL
LIN {X 0,Y 158.255,Z 630.756,A -85,B 0,C 180,E1 -23579.999,E2 -23579.999} C_VEL
LIN {X 0,Y 157.806,Z 630.827,A -85,B 0,C 180,E1 -23587.677,E2 -23587.677} C_VEL
LIN {X 0,Y 157.668,Z 630.829,A -85,B 0,C 180,E1 -23591.3,E2 -23591.3} C_VEL
LIN {X 0,Y 157.449,Z 630.859,A -85,B 0,C 180,E1 -23595.533,E2 -23595.533} C_VEL
LIN {X 0,Y 157.365,Z 630.878,A -85,B 0,C 180,E1 -23600.932,E2 -23600.932} C_VEL
LIN {X 0,Y 157.305,Z 630.87,A -85,B 0,C 180,E1 -23606.68,E2 -23606.68} C_VEL
LIN {X 0,Y 157.272,Z 630.892,A -85,B 0,C 180,E1 -23612.427,E2 -23612.427} C_VEL
LIN {X 0,Y 157.318,Z 630.872,A -85,B 0,C 180,E1 -23616.476,E2 -23616.476} C_VEL
LIN {X 0,Y 157.283,Z 630.89,A -85,B 0,C 180,E1 -23622.085,E2 -23622.085} C_VEL
LIN {X 0,Y 157.292,Z 630.89,A -85,B 0,C 180,E1 -23625.633,E2 -23625.633} C_VEL
LIN {X 0,Y 157.239,Z 630.889,A -85,B 0,C 180,E1 -23631.264,E2 -23631.264} C_VEL
LIN {X 0,Y 157.287,Z 630.894,A -85,B 0,C 180,E1 -23634.489,E2 -23634.489} C_VEL
LIN {X 0,Y 157.29,Z 630.882,A -85,B 0,C 180,E1 -23638.096,E2 -23638.096} C_VEL
LIN {X 0,Y 157.318,Z 630.888,A -85,B 0,C 180,E1 -23643.466,E2 -23643.466} C_VEL
LIN {X 0,Y 157.392,Z 630.877,A -85,B 0,C 180,E1 -23649.666,E2 -23649.666} C_VEL
LIN {X 0,Y 157.482,Z 630.867,A -85,B 0,C 180,E1 -23654.469,E2 -23654.469} C_VEL
LIN {X 0,Y 157.732,Z 630.832,A -85,B 0,C 180,E1 -23659.734,E2 -23659.734} C_VEL
LIN {X 0,Y 157.806,Z 630.822,A -85,B 0,C 180,E1 -23662.322,E2 -23662.322} C_VEL
LIN {X 0,Y 158.255,Z 630.768,A -85,B 0,C 180,E1 -23670,E2 -23670} C_VEL
LIN {X 0,Y 158.071,Z 630.839,A -85,B 0,C 180,E1 -23671.592,E2 -23671.592} C_VEL
LIN {X 0,Y 159.084,Z 633.736,A -85,B 0,C 180,E1 -23672.013,E2 -23672.013} C_VEL
LIN {X 0,Y 168.11,Z 651.592,A -85,B 0,C 180,E1 -23674.993,E2 -23674.993} C_VEL
LIN {X 0,Y 177.471,Z 673.171,A -85,B 0,C 180,E1 -23677.905,E2 -23677.905} C_VEL
LIN {X 0,Y 177.924,Z 674.355,A -85,B 0,C 180,E1 -23678.045,E2 -23678.045} C_VEL
LIN {X 0,Y 174.517,Z 728.073,A -85,B 0,C 180,E1 -23680.501,E2 -23680.501} C_VEL
LIN {X 0,Y 173.072,Z 741.964,A -85,B 0,C 180,E1 -23681.589,E2 -23681.589} C_VEL
LIN {X 0,Y 171.269,Z 754.556,A -85,B 0,C 180,E1 -23683.03,E2 -23683.03} C_VEL
LIN {X 0,Y 169.066,Z 766.831,A -85,B 0,C 180,E1 -23684.946,E2 -23684.946} C_VEL
LIN {X 0,Y 166.585,Z 777.95,A -85,B 0,C 180,E1 -23687.176,E2 -23687.176} C_VEL
LIN {X 0,Y 163.932,Z 789.026,A -85,B 0,C 180,E1 -23690.057,E2 -23690.057} C_VEL
LIN {X 0,Y 161.59,Z 798.109,A -85,B 0,C 180,E1 -23693.043,E2 -23693.043} C_VEL
LIN {X 0,Y 159.548,Z 805.709,A -85,B 0,C 180,E1 -23696.135,E2 -23696.135} C_VEL
LIN {X 0,Y 157.683,Z 813.123,A -85,B 0,C 180,E1 -23699.898,E2 -23699.898} C_VEL
LIN {X 0,Y 156.189,Z 819.51,A -85,B 0,C 180,E1 -23704.103,E2 -23704.103} C_VEL
LIN {X 0,Y 155.258,Z 823.743,A -85,B 0,C 180,E1 -23707.668,E2 -23707.668} C_VEL
LIN {X 0,Y 154.674,Z 827.009,A -85,B 0,C 180,E1 -23711.209,E2 -23711.209} C_VEL
LIN {X 0,Y 154.522,Z 828.532,A -85,B 0,C 180,E1 -23713.307,E2 -23713.307} C_VEL
LIN {X 0,Y 154.596,Z 830.535,A -85,B 0,C 180,E1 -23717.009,E2 -23717.009} C_VEL
LIN {X 0,Y 155.133,Z 831.702,A -85,B 0,C 180,E1 -23720.638,E2 -23720.638} C_VEL
LIN {X 0,Y 156.114,Z 832.116,A -85,B 0,C 180,E1 -23724.182,E2 -23724.182} C_VEL
LIN {X 0,Y 157.629,Z 831.755,A -85,B 0,C 180,E1 -23727.899,E2 -23727.899} C_VEL
LIN {X 0,Y 159.709,Z 830.502,A -85,B 0,C 180,E1 -23731.652,E2 -23731.652} C_VEL
LIN {X 0,Y 162.419,Z 828.321,A -85,B 0,C 180,E1 -23735.321,E2 -23735.321} C_VEL
LIN {X 0,Y 165.72,Z 825.15,A -85,B 0,C 180,E1 -23738.903,E2 -23738.903} C_VEL
LIN {X 0,Y 169.63,Z 820.898,A -85,B 0,C 180,E1 -23742.345,E2 -23742.345} C_VEL
LIN {X 0,Y 174.817,Z 814.629,A -85,B 0,C 180,E1 -23746.043,E2 -23746.043} C_VEL
LIN {X 0,Y 180.317,Z 807.031,A -85,B 0,C 180,E1 -23749.341,E2 -23749.341} C_VEL
LIN {X 0,Y 185.743,Z 798.542,A -85,B 0,C 180,E1 -23752.122,E2 -23752.122} C_VEL
LIN {X 0,Y 191.226,Z 788.44,A -85,B 0,C 180,E1 -23754.643,E2 -23754.643} C_VEL
LIN {X 0,Y 196.537,Z 777.186,A -85,B 0,C 180,E1 -23756.742,E2 -23756.742} C_VEL
LIN {X 0,Y 201.074,Z 765.296,A -85,B 0,C 180,E1 -23758.434,E2 -23758.434} C_VEL
LIN {X 0,Y 204.794,Z 753.063,A -85,B 0,C 180,E1 -23759.745,E2 -23759.745} C_VEL
LIN {X 0,Y 207.564,Z 740.632,A -85,B 0,C 180,E1 -23760.745,E2 -23760.745} C_VEL
LIN {X 0,Y 209.642,Z 727.509,A -85,B 0,C 180,E1 -23761.406,E2 -23761.406} C_VEL
LIN {X 0,Y 212.656,Z 699.262,A -85,B 0,C 180,E1 -23762.459,E2 -23762.459} C_VEL
LIN {X 0,Y 210.435,Z 694.334,A -85,B 0,C 180,E1 -23764.197,E2 -23764.197} C_VEL
LIN {X 0,Y 207.639,Z 688.51,A -85,B 0,C 180,E1 -23766.64,E2 -23766.64} C_VEL
LIN {X 0,Y 206.181,Z 686.231,A -85,B 0,C 180,E1 -23768.053,E2 -23768.053} C_VEL
LIN {X 0,Y 203.763,Z 682.221,A -85,B 0,C 180,E1 -23770.793,E2 -23770.793} C_VEL
LIN {X 0,Y 201.768,Z 679.09,A -85,B 0,C 180,E1 -23773.757,E2 -23773.757} C_VEL
LIN {X 0,Y 199.623,Z 676.23,A -85,B 0,C 180,E1 -23779.422,E2 -23779.422} C_VEL
LIN {X 0,Y 199.413,Z 676.866,A -85,B 0,C 180,E1 -23784.254,E2 -23784.254} C_VEL
LIN {X 0,Y 199.764,Z 678.089,A -85,B 0,C 180,E1 -23786.392,E2 -23786.392} C_VEL
LIN {X 0,Y 202.311,Z 683.518,A -85,B 0,C 180,E1 -23792.059,E2 -23792.059} C_VEL
LIN {X 0,Y 204.815,Z 689.395,A -85,B 0,C 180,E1 -23795.484,E2 -23795.484} C_VEL
LIN {X 0,Y 206.79,Z 694.172,A -85,B 0,C 180,E1 -23797.666,E2 -23797.666} C_VEL
LIN {X 0,Y 209.164,Z 700.122,A -85,B 0,C 180,E1 -23799.87,E2 -23799.87} C_VEL
LIN {X 0,Y 211.831,Z 708.114,A -85,B 0,C 180,E1 -23802.152,E2 -23802.152} C_VEL
LIN {X 0,Y 211.982,Z 709.077,A -85,B 0,C 180,E1 -23802.316,E2 -23802.316} C_VEL
LIN {X 0,Y 208.284,Z 741.543,A -85,B 0,C 180,E1 -23803.505,E2 -23803.505} C_VEL
LIN {X 0,Y 205.657,Z 754.892,A -85,B 0,C 180,E1 -23804.229,E2 -23804.229} C_VEL
LIN {X 0,Y 202.124,Z 767.728,A -85,B 0,C 180,E1 -23805.244,E2 -23805.244} C_VEL
LIN {X 0,Y 197.851,Z 779.628,A -85,B 0,C 180,E1 -23806.511,E2 -23806.511} C_VEL
LIN {X 0,Y 192.729,Z 791.69,A -85,B 0,C 180,E1 -23808.281,E2 -23808.281} C_VEL
LIN {X 0,Y 187.314,Z 802.385,A -85,B 0,C 180,E1 -23810.37,E2 -23810.37} C_VEL
LIN {X 0,Y 182.208,Z 811.183,A -85,B 0,C 180,E1 -23812.592,E2 -23812.592} C_VEL
LIN {X 0,Y 176.668,Z 819.86,A -85,B 0,C 180,E1 -23815.468,E2 -23815.468} C_VEL
LIN {X 0,Y 175.028,Z 822.259,A -85,B 0,C 180,E1 -23816.444,E2 -23816.444} C_VEL
LIN {X 0,Y 172.152,Z 825.575,A -85,B 0,C 180,E1 -23817.753,E2 -23817.753} C_VEL
LIN {X 0,Y 166.062,Z 830.576,A -85,B 0,C 180,E1 -23819.791,E2 -23819.791} C_VEL
LIN {X 0,Y 160.08,Z 834.883,A -85,B 0,C 180,E1 -23822.106,E2 -23822.106} C_VEL
LIN {X 0,Y 157.447,Z 837.092,A -85,B 0,C 180,E1 -23823.832,E2 -23823.832} C_VEL
LIN {X 0,Y 153.341,Z 841.323,A -85,B 0,C 180,E1 -23828.491,E2 -23828.491} C_VEL
LIN {X 0,Y 151.53,Z 842.989,A -85,B 0,C 180,E1 -23831.055,E2 -23831.055} C_VEL
LIN {X 0,Y 150.073,Z 844.248,A -85,B 0,C 180,E1 -23833.681,E2 -23833.681} C_VEL
LIN {X 0,Y 148.369,Z 845.586,A -85,B 0,C 180,E1 -23839.078,E2 -23839.078} C_VEL
LIN {X 0,Y 147.84,Z 845.435,A -85,B 0,C 180,E1 -23844.544,E2 -23844.544} C_VEL
LIN {X 0,Y 147.945,Z 844.755,A -85,B 0,C 180,E1 -23847.277,E2 -23847.277} C_VEL
LIN {X 0,Y 148.179,Z 843.649,A -85,B 0,C 180,E1 -23850,E2 -23850} C_VEL
LIN {X 0,Y 147.993,Z 841.006,A -85,B 0,C 180,E1 -23854.224,E2 -23854.224} C_VEL
LIN {X 0,Y 148.146,Z 837.491,A -85,B 0,C 180,E1 -23858.182,E2 -23858.182} C_VEL
LIN {X 0,Y 148.81,Z 832.684,A -85,B 0,C 180,E1 -23862.27,E2 -23862.27} C_VEL
LIN {X 0,Y 150.034,Z 826.543,A -85,B 0,C 180,E1 -23866.323,E2 -23866.323} C_VEL
LIN {X 0,Y 152.009,Z 818.884,A -85,B 0,C 180,E1 -23870.289,E2 -23870.289} C_VEL
LIN {X 0,Y 154.03,Z 810.992,A -85,B 0,C 180,E1 -23873.53,E2 -23873.53} C_VEL
LIN {X 0,Y 156.661,Z 801.369,A -85,B 0,C 180,E1 -23876.654,E2 -23876.654} C_VEL
LIN {X 0,Y 159.465,Z 790.74,A -85,B 0,C 180,E1 -23879.36,E2 -23879.36} C_VEL
LIN {X 0,Y 162.208,Z 778.879,A -85,B 0,C 180,E1 -23881.69,E2 -23881.69} C_VEL
LIN {X 0,Y 164.858,Z 765.296,A -85,B 0,C 180,E1 -23883.654,E2 -23883.654} C_VEL
LIN {X 0,Y 166.774,Z 752.629,A -85,B 0,C 180,E1 -23884.948,E2 -23884.948} C_VEL
LIN {X 0,Y 168.111,Z 738.777,A -85,B 0,C 180,E1 -23885.881,E2 -23885.881} C_VEL
LIN {X 0,Y 170.518,Z 699.009,A -85,B 0,C 180,E1 -23887.767,E2 -23887.767} C_VEL
LIN {X 0,Y 168.396,Z 678.309,A -85,B 0,C 180,E1 -23889.342,E2 -23889.342} C_VEL
LIN {X 0,Y 160.527,Z 656.394,A -85,B 0,C 180,E1 -23892.19,E2 -23892.19} C_VEL
LIN {X 0,Y 154.072,Z 641.415,A -85,B 0,C 180,E1 -23894.586,E2 -23894.586} C_VEL
LIN {X 0,Y 150.726,Z 633.948,A -85,B 0,C 180,E1 -23895.931,E2 -23895.931} C_VEL
LIN {X 0,Y 150.215,Z 631.775,A -85,B 0,C 180,E1 -23897.497,E2 -23897.497} C_VEL
LIN {X 0,Y 150.23,Z 631.774,A -85,B 0,C 180,E1 -23902.68,E2 -23902.68} C_VEL
LIN {X 0,Y 150.218,Z 631.774,A -85,B 0,C 180,E1 -23907.364,E2 -23907.364} C_VEL
LIN {X 0,Y 150.24,Z 631.767,A -85,B 0,C 180,E1 -23912.719,E2 -23912.719} C_VEL
LIN {X 0,Y 150.348,Z 631.755,A -85,B 0,C 180,E1 -23919.208,E2 -23919.208} C_VEL
LIN {X 0,Y 150.359,Z 631.754,A -85,B 0,C 180,E1 -23923.712,E2 -23923.712} C_VEL
LIN {X 0,Y 150.648,Z 631.708,A -85,B 0,C 180,E1 -23929.244,E2 -23929.244} C_VEL
LIN {X 0,Y 150.735,Z 631.699,A -85,B 0,C 180,E1 -23931.958,E2 -23931.958} C_VEL
LIN {X 0,Y 151.215,Z 631.632,A -85,B 0,C 180,E1 -23939.999,E2 -23939.999} C_VEL
LIN {X 0,Y 150.74,Z 631.706,A -85,B 0,C 180,E1 -23948.039,E2 -23948.039} C_VEL
LIN {X 0,Y 150.602,Z 631.707,A -85,B 0,C 180,E1 -23951.49,E2 -23951.49} C_VEL
LIN {X 0,Y 150.357,Z 631.747,A -85,B 0,C 180,E1 -23956.286,E2 -23956.286} C_VEL
LIN {X 0,Y 150.347,Z 631.752,A -85,B 0,C 180,E1 -23960.791,E2 -23960.791} C_VEL
LIN {X 0,Y 150.237,Z 631.753,A -85,B 0,C 180,E1 -23967.279,E2 -23967.279} C_VEL
LIN {X 0,Y 150.213,Z 631.771,A -85,B 0,C 180,E1 -23972.633,E2 -23972.633} C_VEL
LIN {X 0,Y 150.228,Z 631.75,A -85,B 0,C 180,E1 -23977.456,E2 -23977.456} C_VEL
LIN {X 0,Y 150.224,Z 631.767,A -85,B 0,C 180,E1 -23981.538,E2 -23981.538} C_VEL
LIN {X 0,Y 150.242,Z 631.768,A -85,B 0,C 180,E1 -23985.441,E2 -23985.441} C_VEL
LIN {X 0,Y 150.179,Z 631.759,A -85,B 0,C 180,E1 -23989.069,E2 -23989.069} C_VEL
LIN {X 0,Y 150.213,Z 631.77,A -85,B 0,C 180,E1 -23992.689,E2 -23992.689} C_VEL
LIN {X 0,Y 150.214,Z 631.768,A -85,B 0,C 180,E1 -23997.366,E2 -23997.366} C_VEL
LIN {X 0,Y 150.24,Z 631.77,A -85,B 0,C 180,E1 -24002.718,E2 -24002.718} C_VEL
LIN {X 0,Y 150.349,Z 631.754,A -85,B 0,C 180,E1 -24009.206,E2 -24009.206} C_VEL
LIN {X 0,Y 150.387,Z 631.749,A -85,B 0,C 180,E1 -24013.717,E2 -24013.717} C_VEL
LIN {X 0,Y 150.656,Z 631.713,A -85,B 0,C 180,E1 -24019.246,E2 -24019.246} C_VEL
LIN {X 0,Y 150.742,Z 631.702,A -85,B 0,C 180,E1 -24021.96,E2 -24021.96} C_VEL
LIN {X 0,Y 151.216,Z 631.645,A -85,B 0,C 180,E1 -24030,E2 -24030} C_VEL
LIN {X 0,Y 152.276,Z 634.709,A -85,B 0,C 180,E1 -24030.491,E2 -24030.491} C_VEL
LIN {X 0,Y 162.638,Z 655.401,A -85,B 0,C 180,E1 -24034.147,E2 -24034.147} C_VEL
LIN {X 0,Y 171.57,Z 676.203,A -85,B 0,C 180,E1 -24037.059,E2 -24037.059} C_VEL
LIN {X 0,Y 168.069,Z 728.745,A -85,B 0,C 180,E1 -24039.542,E2 -24039.542} C_VEL
LIN {X 0,Y 166.578,Z 742.252,A -85,B 0,C 180,E1 -24040.637,E2 -24040.637} C_VEL
LIN {X 0,Y 164.658,Z 755.08,A -85,B 0,C 180,E1 -24042.159,E2 -24042.159} C_VEL
LIN {X 0,Y 162.436,Z 766.986,A -85,B 0,C 180,E1 -24044.085,E2 -24044.085} C_VEL
LIN {X 0,Y 159.81,Z 778.375,A -85,B 0,C 180,E1 -24046.455,E2 -24046.455} C_VEL
LIN {X 0,Y 157.129,Z 789.108,A -85,B 0,C 180,E1 -24049.353,E2 -24049.353} C_VEL
LIN {X 0,Y 154.458,Z 798.994,A -85,B 0,C 180,E1 -24052.752,E2 -24052.752} C_VEL
LIN {X 0,Y 152.375,Z 806.498,A -85,B 0,C 180,E1 -24055.986,E2 -24055.986} C_VEL
LIN {X 0,Y 150.723,Z 812.945,A -85,B 0,C 180,E1 -24059.419,E2 -24059.419} C_VEL
LIN {X 0,Y 149.296,Z 818.775,A -85,B 0,C 180,E1 -24063.277,E2 -24063.277} C_VEL
LIN {X 0,Y 148.421,Z 822.548,A -85,B 0,C 180,E1 -24066.394,E2 -24066.394} C_VEL
LIN {X 0,Y 147.664,Z 826.414,A -85,B 0,C 180,E1 -24070.405,E2 -24070.405} C_VEL
LIN {X 0,Y 147.4,Z 829.978,A -85,B 0,C 180,E1 -24075.658,E2 -24075.658} C_VEL
LIN {X 0,Y 147.791,Z 831.577,A -85,B 0,C 180,E1 -24079.538,E2 -24079.538} C_VEL
LIN {X 0,Y 148.724,Z 832.386,A -85,B 0,C 180,E1 -24083.448,E2 -24083.448} C_VEL
LIN {X 0,Y 150.19,Z 832.388,A -85,B 0,C 180,E1 -24087.381,E2 -24087.381} C_VEL
LIN {X 0,Y 153.13,Z 831.001,A -85,B 0,C 180,E1 -24092.682,E2 -24092.682} C_VEL
LIN {X 0,Y 155.642,Z 829.204,A -85,B 0,C 180,E1 -24096.023,E2 -24096.023} C_VEL
LIN {X 0,Y 158.597,Z 826.731,A -85,B 0,C 180,E1 -24099.238,E2 -24099.238} C_VEL
LIN {X 0,Y 163.974,Z 821.464,A -85,B 0,C 180,E1 -24103.868,E2 -24103.868} C_VEL
LIN {X 0,Y 169.334,Z 815.473,A -85,B 0,C 180,E1 -24107.531,E2 -24107.531} C_VEL
LIN {X 0,Y 174.872,Z 808.312,A -85,B 0,C 180,E1 -24110.75,E2 -24110.75} C_VEL
LIN {X 0,Y 180.964,Z 799.403,A -85,B 0,C 180,E1 -24113.747,E2 -24113.747} C_VEL
LIN {X 0,Y 186.51,Z 789.918,A -85,B 0,C 180,E1 -24116.185,E2 -24116.185} C_VEL
LIN {X 0,Y 191.747,Z 779.579,A -85,B 0,C 180,E1 -24118.163,E2 -24118.163} C_VEL
LIN {X 0,Y 196.172,Z 768.983,A -85,B 0,C 180,E1 -24119.771,E2 -24119.771} C_VEL
LIN {X 0,Y 200.197,Z 757.147,A -85,B 0,C 180,E1 -24121.133,E2 -24121.133} C_VEL
LIN {X 0,Y 203.638,Z 743.462,A -85,B 0,C 180,E1 -24122.315,E2 -24122.315} C_VEL
LIN {X 0,Y 206.057,Z 730.105,A -85,B 0,C 180,E1 -24123.043,E2 -24123.043} C_VEL
LIN {X 0,Y 209.223,Z 702.856,A -85,B 0,C 180,E1 -24124.037,E2 -24124.037} C_VEL
LIN {X 0,Y 205.764,Z 695.021,A -85,B 0,C 180,E1 -24127.218,E2 -24127.218} C_VEL
LIN {X 0,Y 203.625,Z 691.619,A -85,B 0,C 180,E1 -24129.443,E2 -24129.443} C_VEL
LIN {X 0,Y 202.032,Z 688.702,A -85,B 0,C 180,E1 -24131.507,E2 -24131.507} C_VEL
LIN {X 0,Y 200.335,Z 685.861,A -85,B 0,C 180,E1 -24134.216,E2 -24134.216} C_VEL
LIN {X 0,Y 198.471,Z 683.243,A -85,B 0,C 180,E1 -24139.539,E2 -24139.539} C_VEL
LIN {X 0,Y 198.249,Z 683.803,A -85,B 0,C 180,E1 -24143.945,E2 -24143.945} C_VEL
LIN {X 0,Y 198.488,Z 684.849,A -85,B 0,C 180,E1 -24145.884,E2 -24145.884} C_VEL
LIN {X 0,Y 200.734,Z 690.182,A -85,B 0,C 180,E1 -24151.469,E2 -24151.469} C_VEL
LIN {X 0,Y 202.9,Z 695.694,A -85,B 0,C 180,E1 -24154.735,E2 -24154.735} C_VEL
LIN {X 0,Y 204.823,Z 700.744,A -85,B 0,C 180,E1 -24157.035,E2 -24157.035} C_VEL
LIN {X 0,Y 206.969,Z 706.76,A -85,B 0,C 180,E1 -24159.212,E2 -24159.212} C_VEL
LIN {X 0,Y 208.458,Z 711.687,A -85,B 0,C 180,E1 -24160.653,E2 -24160.653} C_VEL
LIN {X 0,Y 204.81,Z 742.049,A -85,B 0,C 180,E1 -24161.799,E2 -24161.799} C_VEL
LIN {X 0,Y 202.123,Z 754.998,A -85,B 0,C 180,E1 -24162.498,E2 -24162.498} C_VEL
LIN {X 0,Y 198.524,Z 767.487,A -85,B 0,C 180,E1 -24163.472,E2 -24163.472} C_VEL
LIN {X 0,Y 194.116,Z 779.357,A -85,B 0,C 180,E1 -24164.724,E2 -24164.724} C_VEL
LIN {X 0,Y 188.755,Z 791.37,A -85,B 0,C 180,E1 -24166.465,E2 -24166.465} C_VEL
LIN {X 0,Y 183.071,Z 801.992,A -85,B 0,C 180,E1 -24168.532,E2 -24168.532} C_VEL
LIN {X 0,Y 177.703,Z 810.741,A -85,B 0,C 180,E1 -24170.745,E2 -24170.745} C_VEL
LIN {X 0,Y 171.805,Z 819.442,A -85,B 0,C 180,E1 -24173.62,E2 -24173.62} C_VEL
LIN {X 0,Y 166.479,Z 826.485,A -85,B 0,C 180,E1 -24176.716,E2 -24176.716} C_VEL
LIN {X 0,Y 161.778,Z 832.199,A -85,B 0,C 180,E1 -24180.028,E2 -24180.028} C_VEL
LIN {X 0,Y 157.447,Z 837.092,A -85,B 0,C 180,E1 -24183.832,E2 -24183.832} C_VEL
LIN {X 0,Y 154.903,Z 839.092,A -85,B 0,C 180,E1 -24185.662,E2 -24185.662} C_VEL
LIN {X 0,Y 149.418,Z 841.793,A -85,B 0,C 180,E1 -24188.616,E2 -24188.616} C_VEL
LIN {X 0,Y 144.428,Z 843.682,A -85,B 0,C 180,E1 -24191.864,E2 -24191.864} C_VEL
LIN {X 0,Y 142.726,Z 844.41,A -85,B 0,C 180,E1 -24194.092,E2 -24194.092} C_VEL
LIN {X 0,Y 141.377,Z 845.267,A -85,B 0,C 180,E1 -24198.531,E2 -24198.531} C_VEL
LIN {X 0,Y 140.916,Z 845.307,A -85,B 0,C 180,E1 -24201.395,E2 -24201.395} C_VEL
LIN {X 0,Y 140.827,Z 844.395,A -85,B 0,C 180,E1 -24206.496,E2 -24206.496} C_VEL
LIN {X 0,Y 141.117,Z 843.002,A -85,B 0,C 180,E1 -24210,E2 -24210} C_VEL
LIN {X 0,Y 140.926,Z 840.457,A -85,B 0,C 180,E1 -24214.112,E2 -24214.112} C_VEL
LIN {X 0,Y 141.101,Z 836.549,A -85,B 0,C 180,E1 -24218.593,E2 -24218.593} C_VEL
LIN {X 0,Y 141.849,Z 831.58,A -85,B 0,C 180,E1 -24222.882,E2 -24222.882} C_VEL
LIN {X 0,Y 143.214,Z 825.266,A -85,B 0,C 180,E1 -24227.124,E2 -24227.124} C_VEL
LIN {X 0,Y 144.946,Z 818.785,A -85,B 0,C 180,E1 -24230.58,E2 -24230.58} C_VEL
LIN {X 0,Y 147.014,Z 810.95,A -85,B 0,C 180,E1 -24233.975,E2 -24233.975} C_VEL
LIN {X 0,Y 149.319,Z 803.004,A -85,B 0,C 180,E1 -24236.747,E2 -24236.747} C_VEL
LIN {X 0,Y 152.293,Z 792.186,A -85,B 0,C 180,E1 -24239.741,E2 -24239.741} C_VEL
LIN {X 0,Y 155.054,Z 780.805,A -85,B 0,C 180,E1 -24242.179,E2 -24242.179} C_VEL
LIN {X 0,Y 157.527,Z 769.092,A -85,B 0,C 180,E1 -24244.087,E2 -24244.087} C_VEL
LIN {X 0,Y 159.669,Z 756.487,A -85,B 0,C 180,E1 -24245.579,E2 -24245.579} C_VEL
LIN {X 0,Y 161.347,Z 742.701,A -85,B 0,C 180,E1 -24246.695,E2 -24246.695} C_VEL
LIN {X 0,Y 164.193,Z 699.979,A -85,B 0,C 180,E1 -24248.813,E2 -24248.813} C_VEL
LIN {X 0,Y 162.331,Z 680.839,A -85,B 0,C 180,E1 -24250.308,E2 -24250.308} C_VEL
LIN {X 0,Y 154.977,Z 659.9,A -85,B 0,C 180,E1 -24253.162,E2 -24253.162} C_VEL
LIN {X 0,Y 148.491,Z 644.68,A -85,B 0,C 180,E1 -24255.723,E2 -24255.723} C_VEL
LIN {X 0,Y 144.852,Z 636.991,A -85,B 0,C 180,E1 -24257.213,E2 -24257.213} C_VEL
LIN {X 0,Y 143.361,Z 633.591,A -85,B 0,C 180,E1 -24257.886,E2 -24257.886} C_VEL
LIN {X 0,Y 143.167,Z 632.65,A -85,B 0,C 180,E1 -24258.669,E2 -24258.669} C_VEL
LIN {X 0,Y 143.119,Z 632.659,A -85,B 0,C 180,E1 -24263.893,E2 -24263.893} C_VEL
LIN {X 0,Y 143.185,Z 632.65,A -85,B 0,C 180,E1 -24267.32,E2 -24267.32} C_VEL
LIN {X 0,Y 143.188,Z 632.648,A -85,B 0,C 180,E1 -24272.063,E2 -24272.063} C_VEL
LIN {X 0,Y 143.273,Z 632.639,A -85,B 0,C 180,E1 -24278.746,E2 -24278.746} C_VEL
LIN {X 0,Y 143.298,Z 632.628,A -85,B 0,C 180,E1 -24282.885,E2 -24282.885} C_VEL
LIN {X 0,Y 143.592,Z 632.59,A -85,B 0,C 180,E1 -24288.708,E2 -24288.708} C_VEL
LIN {X 0,Y 143.656,Z 632.577,A -85,B 0,C 180,E1 -24291.559,E2 -24291.559} C_VEL
LIN {X 0,Y 144.174,Z 632.508,A -85,B 0,C 180,E1 -24299.999,E2 -24299.999} C_VEL
LIN {X 0,Y 143.659,Z 632.587,A -85,B 0,C 180,E1 -24308.438,E2 -24308.438} C_VEL
LIN {X 0,Y 143.545,Z 632.584,A -85,B 0,C 180,E1 -24311.711,E2 -24311.711} C_VEL
LIN {X 0,Y 143.297,Z 632.628,A -85,B 0,C 180,E1 -24317.112,E2 -24317.112} C_VEL
LIN {X 0,Y 143.272,Z 632.634,A -85,B 0,C 180,E1 -24321.253,E2 -24321.253} C_VEL
LIN {X 0,Y 143.184,Z 632.634,A -85,B 0,C 180,E1 -24327.934,E2 -24327.934} C_VEL
LIN {X 0,Y 143.164,Z 632.649,A -85,B 0,C 180,E1 -24333.434,E2 -24333.434} C_VEL
LIN {X 0,Y 143.119,Z 632.642,A -85,B 0,C 180,E1 -24339.669,E2 -24339.669} C_VEL
LIN {X 0,Y 143.156,Z 632.652,A -85,B 0,C 180,E1 -24343.415,E2 -24343.415} C_VEL
LIN {X 0,Y 143.13,Z 632.646,A -85,B 0,C 180,E1 -24347.435,E2 -24347.435} C_VEL
LIN {X 0,Y 143.108,Z 632.658,A -85,B 0,C 180,E1 -24353.892,E2 -24353.892} C_VEL
LIN {X 0,Y 143.181,Z 632.644,A -85,B 0,C 180,E1 -24357.322,E2 -24357.322} C_VEL
LIN {X 0,Y 143.186,Z 632.646,A -85,B 0,C 180,E1 -24362.063,E2 -24362.063} C_VEL
LIN {X 0,Y 143.275,Z 632.636,A -85,B 0,C 180,E1 -24368.744,E2 -24368.744} C_VEL
LIN {X 0,Y 143.32,Z 632.629,A -85,B 0,C 180,E1 -24372.889,E2 -24372.889} C_VEL
LIN {X 0,Y 143.591,Z 632.594,A -85,B 0,C 180,E1 -24378.71,E2 -24378.71} C_VEL
LIN {X 0,Y 143.662,Z 632.584,A -85,B 0,C 180,E1 -24381.561,E2 -24381.561} C_VEL
LIN {X 0,Y 143.91,Z 632.555,A -85,B 0,C 180,E1 -24388.127,E2 -24388.127} C_VEL
LIN {X 0,Y 145.142,Z 635.635,A -85,B 0,C 180,E1 -24388.747,E2 -24388.747} C_VEL
LIN {X 0,Y 146.424,Z 637.506,A -85,B 0,C 180,E1 -24389.223,E2 -24389.223} C_VEL
LIN {X 0,Y 157.071,Z 658.904,A -85,B 0,C 180,E1 -24393.195,E2 -24393.195} C_VEL
LIN {X 0,Y 165.138,Z 677.775,A -85,B 0,C 180,E1 -24395.994,E2 -24395.994} C_VEL
LIN {X 0,Y 161.614,Z 729.049,A -85,B 0,C 180,E1 -24398.517,E2 -24398.517} C_VEL
LIN {X 0,Y 160.081,Z 742.433,A -85,B 0,C 180,E1 -24399.635,E2 -24399.635} C_VEL
LIN {X 0,Y 158.084,Z 755.278,A -85,B 0,C 180,E1 -24401.203,E2 -24401.203} C_VEL
LIN {X 0,Y 155.583,Z 768.186,A -85,B 0,C 180,E1 -24403.385,E2 -24403.385} C_VEL
LIN {X 0,Y 152.656,Z 780.141,A -85,B 0,C 180,E1 -24406.035,E2 -24406.035} C_VEL
LIN {X 0,Y 149.871,Z 790.901,A -85,B 0,C 180,E1 -24409.162,E2 -24409.162} C_VEL
LIN {X 0,Y 147.354,Z 799.823,A -85,B 0,C 180,E1 -24412.43,E2 -24412.43} C_VEL
LIN {X 0,Y 144.88,Z 808.51,A -85,B 0,C 180,E1 -24416.481,E2 -24416.481} C_VEL
LIN {X 0,Y 142.86,Z 816.162,A -85,B 0,C 180,E1 -24421.087,E2 -24421.087} C_VEL
LIN {X 0,Y 141.454,Z 822.051,A -85,B 0,C 180,E1 -24425.716,E2 -24425.716} C_VEL
LIN {X 0,Y 140.554,Z 826.604,A -85,B 0,C 180,E1 -24430.542,E2 -24430.542} C_VEL
LIN {X 0,Y 140.293,Z 829.888,A -85,B 0,C 180,E1 -24435.468,E2 -24435.468} C_VEL
LIN {X 0,Y 140.676,Z 831.664,A -85,B 0,C 180,E1 -24439.501,E2 -24439.501} C_VEL
LIN {X 0,Y 141.595,Z 832.656,A -85,B 0,C 180,E1 -24443.446,E2 -24443.446} C_VEL
LIN {X 0,Y 142.95,Z 832.859,A -85,B 0,C 180,E1 -24447.263,E2 -24447.263} C_VEL
LIN {X 0,Y 144.823,Z 832.372,A -85,B 0,C 180,E1 -24450.971,E2 -24450.971} C_VEL
LIN {X 0,Y 147.428,Z 831.051,A -85,B 0,C 180,E1 -24454.92,E2 -24454.92} C_VEL
LIN {X 0,Y 151.918,Z 827.842,A -85,B 0,C 180,E1 -24460.051,E2 -24460.051} C_VEL
LIN {X 0,Y 157.027,Z 823.446,A -85,B 0,C 180,E1 -24464.424,E2 -24464.424} C_VEL
LIN {X 0,Y 162.967,Z 817.365,A -85,B 0,C 180,E1 -24468.526,E2 -24468.526} C_VEL
LIN {X 0,Y 169.392,Z 809.887,A -85,B 0,C 180,E1 -24472.154,E2 -24472.154} C_VEL
LIN {X 0,Y 175.643,Z 801.388,A -85,B 0,C 180,E1 -24475.153,E2 -24475.153} C_VEL
LIN {X 0,Y 181.891,Z 791.483,A -85,B 0,C 180,E1 -24477.787,E2 -24477.787} C_VEL
LIN {X 0,Y 187.271,Z 781.568,A -85,B 0,C 180,E1 -24479.732,E2 -24479.732} C_VEL
LIN {X 0,Y 192.083,Z 770.861,A -85,B 0,C 180,E1 -24481.408,E2 -24481.408} C_VEL
LIN {X 0,Y 196.388,Z 759.218,A -85,B 0,C 180,E1 -24482.782,E2 -24482.782} C_VEL
LIN {X 0,Y 199.905,Z 746.514,A -85,B 0,C 180,E1 -24483.943,E2 -24483.943} C_VEL
LIN {X 0,Y 202.723,Z 732.613,A -85,B 0,C 180,E1 -24484.743,E2 -24484.743} C_VEL
LIN {X 0,Y 205.905,Z 706.607,A -85,B 0,C 180,E1 -24485.715,E2 -24485.715} C_VEL
LIN {X 0,Y 203.463,Z 700.781,A -85,B 0,C 180,E1 -24488.271,E2 -24488.271} C_VEL
LIN {X 0,Y 200.397,Z 695.245,A -85,B 0,C 180,E1 -24492.148,E2 -24492.148} C_VEL
LIN {X 0,Y 199.036,Z 692.75,A -85,B 0,C 180,E1 -24494.507,E2 -24494.507} C_VEL
LIN {X 0,Y 197.319,Z 690.254,A -85,B 0,C 180,E1 -24499.658,E2 -24499.658} C_VEL
LIN {X 0,Y 197.088,Z 690.747,A -85,B 0,C 180,E1 -24503.626,E2 -24503.626} C_VEL
LIN {X 0,Y 197.321,Z 691.892,A -85,B 0,C 180,E1 -24505.758,E2 -24505.758} C_VEL
LIN {X 0,Y 199.219,Z 697.009,A -85,B 0,C 180,E1 -24510.962,E2 -24510.962} C_VEL
LIN {X 0,Y 200.935,Z 701.803,A -85,B 0,C 180,E1 -24513.867,E2 -24513.867} C_VEL
LIN {X 0,Y 202.88,Z 707.272,A -85,B 0,C 180,E1 -24516.366,E2 -24516.366} C_VEL
LIN {X 0,Y 204.773,Z 713.235,A -85,B 0,C 180,E1 -24518.509,E2 -24518.509} C_VEL
LIN {X 0,Y 205.231,Z 714.936,A -85,B 0,C 180,E1 -24519.001,E2 -24519.001} C_VEL
LIN {X 0,Y 201.905,Z 741.025,A -85,B 0,C 180,E1 -24519.935,E2 -24519.935} C_VEL
LIN {X 0,Y 198.916,Z 754.996,A -85,B 0,C 180,E1 -24520.686,E2 -24520.686} C_VEL
LIN {X 0,Y 195.134,Z 767.409,A -85,B 0,C 180,E1 -24521.641,E2 -24521.641} C_VEL
LIN {X 0,Y 190.57,Z 779.144,A -85,B 0,C 180,E1 -24522.866,E2 -24522.866} C_VEL
LIN {X 0,Y 184.982,Z 791.09,A -85,B 0,C 180,E1 -24524.574,E2 -24524.574} C_VEL
LIN {X 0,Y 179.049,Z 801.706,A -85,B 0,C 180,E1 -24526.616,E2 -24526.616} C_VEL
LIN {X 0,Y 173.408,Z 810.447,A -85,B 0,C 180,E1 -24528.809,E2 -24528.809} C_VEL
LIN {X 0,Y 167.158,Z 819.079,A -85,B 0,C 180,E1 -24531.674,E2 -24531.674} C_VEL
LIN {X 0,Y 161.547,Z 826.07,A -85,B 0,C 180,E1 -24534.801,E2 -24534.801} C_VEL
LIN {X 0,Y 155.686,Z 832.619,A -85,B 0,C 180,E1 -24538.727,E2 -24538.727} C_VEL
LIN {X 0,Y 150.944,Z 837.491,A -85,B 0,C 180,E1 -24542.805,E2 -24542.805} C_VEL
LIN {X 0,Y 146.739,Z 841.372,A -85,B 0,C 180,E1 -24547.471,E2 -24547.471} C_VEL
LIN {X 0,Y 143.239,Z 844.071,A -85,B 0,C 180,E1 -24552.88,E2 -24552.88} C_VEL
LIN {X 0,Y 142.726,Z 844.41,A -85,B 0,C 180,E1 -24554.092,E2 -24554.092} C_VEL
LIN {X 0,Y 141.242,Z 844.997,A -85,B 0,C 180,E1 -24556.392,E2 -24556.392} C_VEL
LIN {X 0,Y 137.467,Z 845.118,A -85,B 0,C 180,E1 -24560.167,E2 -24560.167} C_VEL
LIN {X 0,Y 134.281,Z 844.433,A -85,B 0,C 180,E1 -24564.132,E2 -24564.132} C_VEL
LIN {X 0,Y 133.766,Z 843.682,A -85,B 0,C 180,E1 -24566.637,E2 -24566.637} C_VEL
LIN {X 0,Y 134.054,Z 842.336,A -85,B 0,C 180,E1 -24570,E2 -24570} C_VEL
LIN {X 0,Y 133.86,Z 839.889,A -85,B 0,C 180,E1 -24573.99,E2 -24573.99} C_VEL
LIN {X 0,Y 134.066,Z 835.601,A -85,B 0,C 180,E1 -24579.048,E2 -24579.048} C_VEL
LIN {X 0,Y 134.89,Z 830.471,A -85,B 0,C 180,E1 -24583.559,E2 -24583.559} C_VEL
LIN {X 0,Y 136.432,Z 823.931,A -85,B 0,C 180,E1 -24588.003,E2 -24588.003} C_VEL
LIN {X 0,Y 138.681,Z 815.734,A -85,B 0,C 180,E1 -24592.338,E2 -24592.338} C_VEL
LIN {X 0,Y 141.13,Z 807.357,A -85,B 0,C 180,E1 -24595.831,E2 -24595.831} C_VEL
LIN {X 0,Y 144.074,Z 797.081,A -85,B 0,C 180,E1 -24599.196,E2 -24599.196} C_VEL
LIN {X 0,Y 147.191,Z 785.542,A -85,B 0,C 180,E1 -24602.085,E2 -24602.085} C_VEL
LIN {X 0,Y 149.879,Z 774.286,A -85,B 0,C 180,E1 -24604.241,E2 -24604.241} C_VEL
LIN {X 0,Y 152.358,Z 761.677,A -85,B 0,C 180,E1 -24606.024,E2 -24606.024} C_VEL
LIN {X 0,Y 154.269,Z 748.662,A -85,B 0,C 180,E1 -24607.334,E2 -24607.334} C_VEL
LIN {X 0,Y 155.555,Z 735.112,A -85,B 0,C 180,E1 -24608.198,E2 -24608.198} C_VEL
LIN {X 0,Y 157.843,Z 700.367,A -85,B 0,C 180,E1 -24609.957,E2 -24609.957} C_VEL
LIN {X 0,Y 156.169,Z 682.812,A -85,B 0,C 180,E1 -24611.405,E2 -24611.405} C_VEL
LIN {X 0,Y 149.321,Z 663.178,A -85,B 0,C 180,E1 -24614.231,E2 -24614.231} C_VEL
LIN {X 0,Y 143.117,Z 648.402,A -85,B 0,C 180,E1 -24616.832,E2 -24616.832} C_VEL
LIN {X 0,Y 138.062,Z 637.598,A -85,B 0,C 180,E1 -24619.064,E2 -24619.064} C_VEL
LIN {X 0,Y 136.373,Z 634.884,A -85,B 0,C 180,E1 -24619.777,E2 -24619.777} C_VEL
LIN {X 0,Y 136.083,Z 633.535,A -85,B 0,C 180,E1 -24620.002,E2 -24620.002} C_VEL
LIN {X 0,Y 136.091,Z 633.534,A -85,B 0,C 180,E1 -24625.715,E2 -24625.715} C_VEL
LIN {X 0,Y 136.143,Z 633.526,A -85,B 0,C 180,E1 -24632.314,E2 -24632.314} C_VEL
LIN {X 0,Y 136.24,Z 633.515,A -85,B 0,C 180,E1 -24638.831,E2 -24638.831} C_VEL
LIN {X 0,Y 136.269,Z 633.512,A -85,B 0,C 180,E1 -24645.055,E2 -24645.055} C_VEL
LIN {X 0,Y 136.495,Z 633.479,A -85,B 0,C 180,E1 -24648.113,E2 -24648.113} C_VEL
LIN {X 0,Y 136.584,Z 633.455,A -85,B 0,C 180,E1 -24651.118,E2 -24651.118} C_VEL
LIN {X 0,Y 137.131,Z 633.385,A -85,B 0,C 180,E1 -24659.999,E2 -24659.999} C_VEL
LIN {X 0,Y 136.587,Z 633.468,A -85,B 0,C 180,E1 -24668.878,E2 -24668.878} C_VEL
LIN {X 0,Y 136.488,Z 633.461,A -85,B 0,C 180,E1 -24671.953,E2 -24671.953} C_VEL
LIN {X 0,Y 136.237,Z 633.511,A -85,B 0,C 180,E1 -24678.029,E2 -24678.029} C_VEL
LIN {X 0,Y 136.193,Z 633.512,A -85,B 0,C 180,E1 -24681.747,E2 -24681.747} C_VEL
LIN {X 0,Y 136.094,Z 633.521,A -85,B 0,C 180,E1 -24688.614,E2 -24688.614} C_VEL
LIN {X 0,Y 136.078,Z 633.526,A -85,B 0,C 180,E1 -24694.617,E2 -24694.617} C_VEL
LIN {X 0,Y 136.085,Z 633.513,A -85,B 0,C 180,E1 -24699.227,E2 -24699.227} C_VEL
LIN {X 0,Y 136.09,Z 633.532,A -85,B 0,C 180,E1 -24703.7,E2 -24703.7} C_VEL
LIN {X 0,Y 136.081,Z 633.52,A -85,B 0,C 180,E1 -24707.826,E2 -24707.826} C_VEL
LIN {X 0,Y 136.06,Z 633.528,A -85,B 0,C 180,E1 -24711.696,E2 -24711.696} C_VEL
LIN {X 0,Y 136.086,Z 633.533,A -85,B 0,C 180,E1 -24715.718,E2 -24715.718} C_VEL
LIN {X 0,Y 136.143,Z 633.524,A -85,B 0,C 180,E1 -24722.316,E2 -24722.316} C_VEL
LIN {X 0,Y 136.242,Z 633.512,A -85,B 0,C 180,E1 -24728.833,E2 -24728.833} C_VEL
LIN {X 0,Y 136.284,Z 633.506,A -85,B 0,C 180,E1 -24735.058,E2 -24735.058} C_VEL
LIN {X 0,Y 136.494,Z 633.479,A -85,B 0,C 180,E1 -24738.115,E2 -24738.115} C_VEL
LIN {X 0,Y 136.589,Z 633.466,A -85,B 0,C 180,E1 -24741.121,E2 -24741.121} C_VEL
LIN {X 0,Y 136.682,Z 633.455,A -85,B 0,C 180,E1 -24746.13,E2 -24746.13} C_VEL
LIN {X 0,Y 137.738,Z 636.294,A -85,B 0,C 180,E1 -24746.7,E2 -24746.7} C_VEL
LIN {X 0,Y 139.372,Z 638.496,A -85,B 0,C 180,E1 -24747.346,E2 -24747.346} C_VEL
LIN {X 0,Y 142.738,Z 644.393,A -85,B 0,C 180,E1 -24748.74,E2 -24748.74} C_VEL
LIN {X 0,Y 151.677,Z 662.779,A -85,B 0,C 180,E1 -24752.258,E2 -24752.258} C_VEL
LIN {X 0,Y 158.863,Z 679.622,A -85,B 0,C 180,E1 -24754.898,E2 -24754.898} C_VEL
LIN {X 0,Y 155.205,Z 729.602,A -85,B 0,C 180,E1 -24757.429,E2 -24757.429} C_VEL
LIN {X 0,Y 153.636,Z 742.621,A -85,B 0,C 180,E1 -24758.55,E2 -24758.55} C_VEL
LIN {X 0,Y 151.542,Z 755.599,A -85,B 0,C 180,E1 -24760.184,E2 -24760.184} C_VEL
LIN {X 0,Y 149.047,Z 768.001,A -85,B 0,C 180,E1 -24762.343,E2 -24762.343} C_VEL
LIN {X 0,Y 146.059,Z 779.857,A -85,B 0,C 180,E1 -24765.029,E2 -24765.029} C_VEL
LIN {X 0,Y 143.196,Z 790.574,A -85,B 0,C 180,E1 -24768.233,E2 -24768.233} C_VEL
LIN {X 0,Y 140.252,Z 800.63,A -85,B 0,C 180,E1 -24772.075,E2 -24772.075} C_VEL
LIN {X 0,Y 138.015,Z 808.214,A -85,B 0,C 180,E1 -24775.772,E2 -24775.772} C_VEL
LIN {X 0,Y 136.083,Z 815.079,A -85,B 0,C 180,E1 -24779.977,E2 -24779.977} C_VEL
LIN {X 0,Y 134.505,Z 821.538,A -85,B 0,C 180,E1 -24785.082,E2 -24785.082} C_VEL
LIN {X 0,Y 133.659,Z 825.463,A -85,B 0,C 180,E1 -24789.121,E2 -24789.121} C_VEL
LIN {X 0,Y 133.221,Z 828.602,A -85,B 0,C 180,E1 -24793.298,E2 -24793.298} C_VEL
LIN {X 0,Y 133.318,Z 830.949,A -85,B 0,C 180,E1 -24797.562,E2 -24797.562} C_VEL
LIN {X 0,Y 134.04,Z 832.478,A -85,B 0,C 180,E1 -24801.856,E2 -24801.856} C_VEL
LIN {X 0,Y 135.352,Z 833.189,A -85,B 0,C 180,E1 -24806.177,E2 -24806.177} C_VEL
LIN {X 0,Y 137.282,Z 833.09,A -85,B 0,C 180,E1 -24810.491,E2 -24810.491} C_VEL
LIN {X 0,Y 139.929,Z 832.146,A -85,B 0,C 180,E1 -24814.693,E2 -24814.693} C_VEL
LIN {X 0,Y 144.449,Z 829.509,A -85,B 0,C 180,E1 -24820.089,E2 -24820.089} C_VEL
LIN {X 0,Y 148.081,Z 826.843,A -85,B 0,C 180,E1 -24823.457,E2 -24823.457} C_VEL
LIN {X 0,Y 153.309,Z 822.442,A -85,B 0,C 180,E1 -24827.425,E2 -24827.425} C_VEL
LIN {X 0,Y 159.478,Z 816.492,A -85,B 0,C 180,E1 -24831.197,E2 -24831.197} C_VEL
LIN {X 0,Y 164.959,Z 810.303,A -85,B 0,C 180,E1 -24834.135,E2 -24834.135} C_VEL
LIN {X 0,Y 171.914,Z 801.33,A -85,B 0,C 180,E1 -24837.265,E2 -24837.265} C_VEL
LIN {X 0,Y 178.072,Z 792.082,A -85,B 0,C 180,E1 -24839.708,E2 -24839.708} C_VEL
LIN {X 0,Y 183.601,Z 782.472,A -85,B 0,C 180,E1 -24841.593,E2 -24841.593} C_VEL
LIN {X 0,Y 188.859,Z 771.279,A -85,B 0,C 180,E1 -24843.32,E2 -24843.32} C_VEL
LIN {X 0,Y 193.374,Z 759.47,A -85,B 0,C 180,E1 -24844.692,E2 -24844.692} C_VEL
LIN {X 0,Y 197.122,Z 746.438,A -85,B 0,C 180,E1 -24845.84,E2 -24845.84} C_VEL
LIN {X 0,Y 199.937,Z 733.076,A -85,B 0,C 180,E1 -24846.595,E2 -24846.595} C_VEL
LIN {X 0,Y 202.859,Z 710.65,A -85,B 0,C 180,E1 -24847.423,E2 -24847.423} C_VEL
LIN {X 0,Y 201.333,Z 706.707,A -85,B 0,C 180,E1 -24849.237,E2 -24849.237} C_VEL
LIN {X 0,Y 198.811,Z 701.856,A -85,B 0,C 180,E1 -24852.756,E2 -24852.756} C_VEL
LIN {X 0,Y 197.547,Z 699.403,A -85,B 0,C 180,E1 -24855.212,E2 -24855.212} C_VEL
LIN {X 0,Y 196.169,Z 697.266,A -85,B 0,C 180,E1 -24859.778,E2 -24859.778} C_VEL
LIN {X 0,Y 195.973,Z 697.813,A -85,B 0,C 180,E1 -24863.769,E2 -24863.769} C_VEL
LIN {X 0,Y 196.319,Z 699.695,A -85,B 0,C 180,E1 -24866.498,E2 -24866.498} C_VEL
LIN {X 0,Y 197.695,Z 703.698,A -85,B 0,C 180,E1 -24870.385,E2 -24870.385} C_VEL
LIN {X 0,Y 199.198,Z 708.249,A -85,B 0,C 180,E1 -24873.151,E2 -24873.151} C_VEL
LIN {X 0,Y 201.009,Z 713.892,A -85,B 0,C 180,E1 -24875.738,E2 -24875.738} C_VEL
LIN {X 0,Y 202.124,Z 718.086,A -85,B 0,C 180,E1 -24877.213,E2 -24877.213} C_VEL
LIN {X 0,Y 199.023,Z 741.296,A -85,B 0,C 180,E1 -24878.088,E2 -24878.088} C_VEL
LIN {X 0,Y 195.866,Z 755.286,A -85,B 0,C 180,E1 -24878.827,E2 -24878.827} C_VEL
LIN {X 0,Y 191.966,Z 767.517,A -85,B 0,C 180,E1 -24879.753,E2 -24879.753} C_VEL
LIN {X 0,Y 187.246,Z 779.171,A -85,B 0,C 180,E1 -24880.945,E2 -24880.945} C_VEL
LIN {X 0,Y 181.44,Z 790.983,A -85,B 0,C 180,E1 -24882.614,E2 -24882.614} C_VEL
LIN {X 0,Y 175.246,Z 801.489,A -85,B 0,C 180,E1 -24884.617,E2 -24884.617} C_VEL
LIN {X 0,Y 168.209,Z 811.743,A -85,B 0,C 180,E1 -24887.24,E2 -24887.24} C_VEL
LIN {X 0,Y 161.702,Z 820.018,A -85,B 0,C 180,E1 -24890.129,E2 -24890.129} C_VEL
LIN {X 0,Y 155.825,Z 826.762,A -85,B 0,C 180,E1 -24893.303,E2 -24893.303} C_VEL
LIN {X 0,Y 149.673,Z 833.061,A -85,B 0,C 180,E1 -24897.318,E2 -24897.318} C_VEL
LIN {X 0,Y 145.182,Z 837.272,A -85,B 0,C 180,E1 -24901.049,E2 -24901.049} C_VEL
LIN {X 0,Y 142.467,Z 839.56,A -85,B 0,C 180,E1 -24903.643,E2 -24903.643} C_VEL
LIN {X 0,Y 138.128,Z 842.835,A -85,B 0,C 180,E1 -24909.136,E2 -24909.136} C_VEL
LIN {X 0,Y 135.739,Z 844.297,A -85,B 0,C 180,E1 -24913.633,E2 -24913.633} C_VEL
LIN {X 0,Y 134.41,Z 844.935,A -85,B 0,C 180,E1 -24917.928,E2 -24917.928} C_VEL
LIN {X 0,Y 133.699,Z 844.401,A -85,B 0,C 180,E1 -24923.965,E2 -24923.965} C_VEL
LIN {X 0,Y 133.766,Z 843.682,A -85,B 0,C 180,E1 -24926.637,E2 -24926.637} C_VEL
LIN {X 0,Y 133.586,Z 843.056,A -85,B 0,C 180,E1 -24928.294,E2 -24928.294} C_VEL
LIN {X 0,Y 132.304,Z 841.788,A -85,B 0,C 180,E1 -24930.724,E2 -24930.724} C_VEL
LIN {X 0,Y 129.099,Z 838.95,A -85,B 0,C 180,E1 -24934.707,E2 -24934.707} C_VEL
LIN {X 0,Y 127.228,Z 836.084,A -85,B 0,C 180,E1 -24937.988,E2 -24937.988} C_VEL
LIN {X 0,Y 127.072,Z 834.458,A -85,B 0,C 180,E1 -24939.649,E2 -24939.649} C_VEL
LIN {X 0,Y 128.206,Z 828.201,A -85,B 0,C 180,E1 -24945.093,E2 -24945.093} C_VEL
LIN {X 0,Y 130.072,Z 821.243,A -85,B 0,C 180,E1 -24949.736,E2 -24949.736} C_VEL
LIN {X 0,Y 132.059,Z 814.066,A -85,B 0,C 180,E1 -24953.524,E2 -24953.524} C_VEL
LIN {X 0,Y 134.761,Z 805.418,A -85,B 0,C 180,E1 -24957.15,E2 -24957.15} C_VEL
LIN {X 0,Y 137.913,Z 794.757,A -85,B 0,C 180,E1 -24960.636,E2 -24960.636} C_VEL
LIN {X 0,Y 140.802,Z 784.242,A -85,B 0,C 180,E1 -24963.301,E2 -24963.301} C_VEL
LIN {X 0,Y 143.622,Z 772.7,A -85,B 0,C 180,E1 -24965.526,E2 -24965.526} C_VEL
LIN {X 0,Y 146.2,Z 759.72,A -85,B 0,C 180,E1 -24967.364,E2 -24967.364} C_VEL
LIN {X 0,Y 148.056,Z 747.107,A -85,B 0,C 180,E1 -24968.622,E2 -24968.622} C_VEL
LIN {X 0,Y 149.532,Z 730.672,A -85,B 0,C 180,E1 -24969.624,E2 -24969.624} C_VEL
LIN {X 0,Y 151.549,Z 700.791,A -85,B 0,C 180,E1 -24971.196,E2 -24971.196} C_VEL
LIN {X 0,Y 150.056,Z 684.832,A -85,B 0,C 180,E1 -24972.59,E2 -24972.59} C_VEL
LIN {X 0,Y 143.885,Z 666.873,A -85,B 0,C 180,E1 -24975.276,E2 -24975.276} C_VEL
LIN {X 0,Y 136.841,Z 649.743,A -85,B 0,C 180,E1 -24978.481,E2 -24978.481} C_VEL
LIN {X 0,Y 132.821,Z 641.663,A -85,B 0,C 180,E1 -24980.335,E2 -24980.335} C_VEL
LIN {X 0,Y 130.682,Z 638.146,A -85,B 0,C 180,E1 -24981.322,E2 -24981.322} C_VEL
LIN {X 0,Y 129.245,Z 635.493,A -85,B 0,C 180,E1 -24982.036,E2 -24982.036} C_VEL
LIN {X 0,Y 129.015,Z 634.415,A -85,B 0,C 180,E1 -24982.265,E2 -24982.265} C_VEL
LIN {X 0,Y 128.996,Z 634.419,A -85,B 0,C 180,E1 -24986.986,E2 -24986.986} C_VEL
LIN {X 0,Y 129.016,Z 634.413,A -85,B 0,C 180,E1 -24990.64,E2 -24990.64} C_VEL
LIN {X 0,Y 129.026,Z 634.404,A -85,B 0,C 180,E1 -24994.165,E2 -24994.165} C_VEL
LIN {X 0,Y 129.106,Z 634.405,A -85,B 0,C 180,E1 -24997.727,E2 -24997.727} C_VEL
LIN {X 0,Y 129.186,Z 634.393,A -85,B 0,C 180,E1 -25004.214,E2 -25004.214} C_VEL
LIN {X 0,Y 129.414,Z 634.361,A -85,B 0,C 180,E1 -25007.819,E2 -25007.819} C_VEL
LIN {X 0,Y 129.511,Z 634.335,A -85,B 0,C 180,E1 -25010.629,E2 -25010.629} C_VEL
LIN {X 0,Y 130.086,Z 634.261,A -85,B 0,C 180,E1 -25019.998,E2 -25019.998} C_VEL
LIN {X 0,Y 129.513,Z 634.345,A -85,B 0,C 180,E1 -25029.368,E2 -25029.368} C_VEL
LIN {X 0,Y 129.389,Z 634.341,A -85,B 0,C 180,E1 -25032.547,E2 -25032.547} C_VEL
LIN {X 0,Y 129.149,Z 634.394,A -85,B 0,C 180,E1 -25039.055,E2 -25039.055} C_VEL
LIN {X 0,Y 129.104,Z 634.392,A -85,B 0,C 180,E1 -25042.397,E2 -25042.397} C_VEL
LIN {X 0,Y 129.024,Z 634.385,A -85,B 0,C 180,E1 -25045.832,E2 -25045.832} C_VEL
LIN {X 0,Y 129.013,Z 634.406,A -85,B 0,C 180,E1 -25049.357,E2 -25049.357} C_VEL
LIN {X 0,Y 129.02,Z 634.402,A -85,B 0,C 180,E1 -25055.208,E2 -25055.208} C_VEL
LIN {X 0,Y 129.01,Z 634.404,A -85,B 0,C 180,E1 -25060.82,E2 -25060.82} C_VEL
LIN {X 0,Y 129.019,Z 634.412,A -85,B 0,C 180,E1 -25065.082,E2 -25065.082} C_VEL
LIN {X 0,Y 128.993,Z 634.395,A -85,B 0,C 180,E1 -25069.706,E2 -25069.706} C_VEL
LIN {X 0,Y 128.99,Z 634.418,A -85,B 0,C 180,E1 -25074.81,E2 -25074.81} C_VEL
LIN {X 0,Y 129.013,Z 634.402,A -85,B 0,C 180,E1 -25080.642,E2 -25080.642} C_VEL
LIN {X 0,Y 129.027,Z 634.413,A -85,B 0,C 180,E1 -25084.167,E2 -25084.167} C_VEL
LIN {X 0,Y 129.104,Z 634.403,A -85,B 0,C 180,E1 -25087.727,E2 -25087.727} C_VEL
LIN {X 0,Y 129.161,Z 634.396,A -85,B 0,C 180,E1 -25090.945,E2 -25090.945} C_VEL
LIN {X 0,Y 129.413,Z 634.361,A -85,B 0,C 180,E1 -25097.82,E2 -25097.82} C_VEL
LIN {X 0,Y 129.515,Z 634.348,A -85,B 0,C 180,E1 -25100.631,E2 -25100.631} C_VEL
LIN {X 0,Y 129.535,Z 634.45,A -85,B 0,C 180,E1 -25103.946,E2 -25103.946} C_VEL
LIN {X 0,Y 130.521,Z 637.168,A -85,B 0,C 180,E1 -25104.515,E2 -25104.515} C_VEL
LIN {X 0,Y 132.168,Z 639.471,A -85,B 0,C 180,E1 -25105.25,E2 -25105.25} C_VEL
LIN {X 0,Y 137.352,Z 647.861,A -85,B 0,C 180,E1 -25107.497,E2 -25107.497} C_VEL
LIN {X 0,Y 146.541,Z 667.182,A -85,B 0,C 180,E1 -25111.366,E2 -25111.366} C_VEL
LIN {X 0,Y 152.53,Z 681.66,A -85,B 0,C 180,E1 -25113.704,E2 -25113.704} C_VEL
LIN {X 0,Y 148.781,Z 730.154,A -85,B 0,C 180,E1 -25116.253,E2 -25116.253} C_VEL
LIN {X 0,Y 147.119,Z 743.92,A -85,B 0,C 180,E1 -25117.52,E2 -25117.52} C_VEL
LIN {X 0,Y 144.858,Z 756.819,A -85,B 0,C 180,E1 -25119.248,E2 -25119.248} C_VEL
LIN {X 0,Y 142.375,Z 768.529,A -85,B 0,C 180,E1 -25121.388,E2 -25121.388} C_VEL
LIN {X 0,Y 139.212,Z 780.544,A -85,B 0,C 180,E1 -25124.247,E2 -25124.247} C_VEL
LIN {X 0,Y 136.164,Z 791.442,A -85,B 0,C 180,E1 -25127.686,E2 -25127.686} C_VEL
LIN {X 0,Y 133.15,Z 801.311,A -85,B 0,C 180,E1 -25131.683,E2 -25131.683} C_VEL
LIN {X 0,Y 130.462,Z 810.197,A -85,B 0,C 180,E1 -25136.386,E2 -25136.386} C_VEL
LIN {X 0,Y 128.483,Z 817.395,A -85,B 0,C 180,E1 -25141.306,E2 -25141.306} C_VEL
LIN {X 0,Y 127.187,Z 822.501,A -85,B 0,C 180,E1 -25145.8,E2 -25145.8} C_VEL
LIN {X 0,Y 126.376,Z 826.517,A -85,B 0,C 180,E1 -25150.34,E2 -25150.34} C_VEL
LIN {X 0,Y 126.127,Z 830.362,A -85,B 0,C 180,E1 -25156.416,E2 -25156.416} C_VEL
LIN {X 0,Y 127.06,Z 832.718,A -85,B 0,C 180,E1 -25162.525,E2 -25162.525} C_VEL
LIN {X 0,Y 128.404,Z 833.505,A -85,B 0,C 180,E1 -25166.818,E2 -25166.818} C_VEL
LIN {X 0,Y 130.266,Z 833.602,A -85,B 0,C 180,E1 -25170.953,E2 -25170.953} C_VEL
LIN {X 0,Y 132.757,Z 832.951,A -85,B 0,C 180,E1 -25174.945,E2 -25174.945} C_VEL
LIN {X 0,Y 135.72,Z 831.646,A -85,B 0,C 180,E1 -25178.761,E2 -25178.761} C_VEL
LIN {X 0,Y 139.734,Z 829.336,A -85,B 0,C 180,E1 -25182.861,E2 -25182.861} C_VEL
LIN {X 0,Y 146.01,Z 824.81,A -85,B 0,C 180,E1 -25187.88,E2 -25187.88} C_VEL
LIN {X 0,Y 152.693,Z 819.05,A -85,B 0,C 180,E1 -25192.065,E2 -25192.065} C_VEL
LIN {X 0,Y 160.176,Z 811.416,A -85,B 0,C 180,E1 -25195.942,E2 -25195.942} C_VEL
LIN {X 0,Y 166.559,Z 803.903,A -85,B 0,C 180,E1 -25198.697,E2 -25198.697} C_VEL
LIN {X 0,Y 172.941,Z 795.064,A -85,B 0,C 180,E1 -25201.167,E2 -25201.167} C_VEL
LIN {X 0,Y 179.623,Z 784.253,A -85,B 0,C 180,E1 -25203.366,E2 -25203.366} C_VEL
LIN {X 0,Y 185.248,Z 773.215,A -85,B 0,C 180,E1 -25205.105,E2 -25205.105} C_VEL
LIN {X 0,Y 190.365,Z 760.662,A -85,B 0,C 180,E1 -25206.579,E2 -25206.579} C_VEL
LIN {X 0,Y 194.391,Z 747.603,A -85,B 0,C 180,E1 -25207.726,E2 -25207.726} C_VEL
LIN {X 0,Y 197.377,Z 734.082,A -85,B 0,C 180,E1 -25208.485,E2 -25208.485} C_VEL
LIN {X 0,Y 200.024,Z 714.469,A -85,B 0,C 180,E1 -25209.245,E2 -25209.245} C_VEL
LIN {X 0,Y 199.009,Z 712.193,A -85,B 0,C 180,E1 -25210.58,E2 -25210.58} C_VEL
LIN {X 0,Y 197.231,Z 708.427,A -85,B 0,C 180,E1 -25213.403,E2 -25213.403} C_VEL
LIN {X 0,Y 196.26,Z 706.317,A -85,B 0,C 180,E1 -25215.517,E2 -25215.517} C_VEL
LIN {X 0,Y 195.093,Z 704.362,A -85,B 0,C 180,E1 -25219.448,E2 -25219.448} C_VEL
LIN {X 0,Y 194.786,Z 704.612,A -85,B 0,C 180,E1 -25222.94,E2 -25222.94} C_VEL
LIN {X 0,Y 194.898,Z 705.366,A -85,B 0,C 180,E1 -25224.618,E2 -25224.618} C_VEL
LIN {X 0,Y 196.068,Z 709.76,A -85,B 0,C 180,E1 -25229.379,E2 -25229.379} C_VEL
LIN {X 0,Y 197.414,Z 714.452,A -85,B 0,C 180,E1 -25232.277,E2 -25232.277} C_VEL
LIN {X 0,Y 198.93,Z 719.89,A -85,B 0,C 180,E1 -25234.801,E2 -25234.801} C_VEL
LIN {X 0,Y 199.368,Z 721.876,A -85,B 0,C 180,E1 -25235.481,E2 -25235.481} C_VEL
LIN {X 0,Y 196.441,Z 741.909,A -85,B 0,C 180,E1 -25236.184,E2 -25236.184} C_VEL
LIN {X 0,Y 193.267,Z 755.127,A -85,B 0,C 180,E1 -25236.871,E2 -25236.871} C_VEL
LIN {X 0,Y 189.025,Z 767.793,A -85,B 0,C 180,E1 -25237.809,E2 -25237.809} C_VEL
LIN {X 0,Y 184.144,Z 779.252,A -85,B 0,C 180,E1 -25238.958,E2 -25238.958} C_VEL
LIN {X 0,Y 178.118,Z 790.923,A -85,B 0,C 180,E1 -25240.578,E2 -25240.578} C_VEL
LIN {X 0,Y 171.691,Z 801.384,A -85,B 0,C 180,E1 -25242.541,E2 -25242.541} C_VEL
LIN {X 0,Y 165.494,Z 810.014,A -85,B 0,C 180,E1 -25244.659,E2 -25244.659} C_VEL
LIN {X 0,Y 158.632,Z 818.517,A -85,B 0,C 180,E1 -25247.498,E2 -25247.498} C_VEL
LIN {X 0,Y 152.27,Z 825.431,A -85,B 0,C 180,E1 -25250.609,E2 -25250.609} C_VEL
LIN {X 0,Y 145.503,Z 831.923,A -85,B 0,C 180,E1 -25254.577,E2 -25254.577} C_VEL
LIN {X 0,Y 140.982,Z 835.903,A -85,B 0,C 180,E1 -25257.938,E2 -25257.938} C_VEL
LIN {X 0,Y 136.142,Z 839.658,A -85,B 0,C 180,E1 -25262.316,E2 -25262.316} C_VEL
LIN {X 0,Y 131.5,Z 842.758,A -85,B 0,C 180,E1 -25268.031,E2 -25268.031} C_VEL
LIN {X 0,Y 129.676,Z 843.744,A -85,B 0,C 180,E1 -25271.024,E2 -25271.024} C_VEL
LIN {X 0,Y 127.438,Z 844.543,A -85,B 0,C 180,E1 -25277.256,E2 -25277.256} C_VEL
LIN {X 0,Y 126.628,Z 843.868,A -85,B 0,C 180,E1 -25283.627,E2 -25283.627} C_VEL
LIN {X 0,Y 126.722,Z 842.962,A -85,B 0,C 180,E1 -25286.821,E2 -25286.821} C_VEL
LIN {X 0,Y 126.993,Z 841.607,A -85,B 0,C 180,E1 -25290,E2 -25290} C_VEL
LIN {X 0,Y 126.8,Z 839.268,A -85,B 0,C 180,E1 -25293.892,E2 -25293.892} C_VEL
LIN {X 0,Y 127.06,Z 834.557,A -85,B 0,C 180,E1 -25299.551,E2 -25299.551} C_VEL
LIN {X 0,Y 127.072,Z 834.458,A -85,B 0,C 180,E1 -25299.649,E2 -25299.649} C_VEL
LIN {X 0,Y 126.8,Z 831.904,A -85,B 0,C 180,E1 -25302.036,E2 -25302.036} C_VEL
LIN {X 0,Y 124.939,Z 827.093,A -85,B 0,C 180,E1 -25305.887,E2 -25305.887} C_VEL
LIN {X 0,Y 123.49,Z 821.594,A -85,B 0,C 180,E1 -25309.67,E2 -25309.67} C_VEL
LIN {X 0,Y 123.876,Z 817.962,A -85,B 0,C 180,E1 -25311.852,E2 -25311.852} C_VEL
LIN {X 0,Y 126.595,Z 808.874,A -85,B 0,C 180,E1 -25316.367,E2 -25316.367} C_VEL
LIN {X 0,Y 129.655,Z 799.366,A -85,B 0,C 180,E1 -25320.001,E2 -25320.001} C_VEL
LIN {X 0,Y 132.956,Z 788.385,A -85,B 0,C 180,E1 -25323.258,E2 -25323.258} C_VEL
LIN {X 0,Y 136.182,Z 776.259,A -85,B 0,C 180,E1 -25325.946,E2 -25325.946} C_VEL
LIN {X 0,Y 139.026,Z 763.532,A -85,B 0,C 180,E1 -25328.031,E2 -25328.031} C_VEL
LIN {X 0,Y 141.183,Z 750.711,A -85,B 0,C 180,E1 -25329.511,E2 -25329.511} C_VEL
LIN {X 0,Y 142.76,Z 737.071,A -85,B 0,C 180,E1 -25330.535,E2 -25330.535} C_VEL
LIN {X 0,Y 145.325,Z 701.456,A -85,B 0,C 180,E1 -25332.479,E2 -25332.479} C_VEL
LIN {X 0,Y 143.975,Z 686.841,A -85,B 0,C 180,E1 -25333.817,E2 -25333.817} C_VEL
LIN {X 0,Y 137.941,Z 669.148,A -85,B 0,C 180,E1 -25336.666,E2 -25336.666} C_VEL
LIN {X 0,Y 132.213,Z 655.031,A -85,B 0,C 180,E1 -25339.431,E2 -25339.431} C_VEL
LIN {X 0,Y 128.273,Z 646.535,A -85,B 0,C 180,E1 -25341.409,E2 -25341.409} C_VEL
LIN {X 0,Y 124.007,Z 639.503,A -85,B 0,C 180,E1 -25343.558,E2 -25343.558} C_VEL
LIN {X 0,Y 122.354,Z 636.962,A -85,B 0,C 180,E1 -25344.404,E2 -25344.404} C_VEL
LIN {X 0,Y 121.969,Z 635.291,A -85,B 0,C 180,E1 -25344.813,E2 -25344.813} C_VEL
LIN {X 0,Y 121.929,Z 635.293,A -85,B 0,C 180,E1 -25349.835,E2 -25349.835} C_VEL
LIN {X 0,Y 121.981,Z 635.289,A -85,B 0,C 180,E1 -25356.213,E2 -25356.213} C_VEL
LIN {X 0,Y 122.032,Z 635.28,A -85,B 0,C 180,E1 -25359.783,E2 -25359.783} C_VEL
LIN {X 0,Y 122.361,Z 635.241,A -85,B 0,C 180,E1 -25367.526,E2 -25367.526} C_VEL
LIN {X 0,Y 122.442,Z 635.216,A -85,B 0,C 180,E1 -25370.083,E2 -25370.083} C_VEL
LIN {X 0,Y 122.602,Z 635.213,A -85,B 0,C 180,E1 -25376.712,E2 -25376.712} C_VEL
LIN {X 0,Y 123.04,Z 635.138,A -85,B 0,C 180,E1 -25379.998,E2 -25379.998} C_VEL
LIN {X 0,Y 122.415,Z 635.23,A -85,B 0,C 180,E1 -25387.135,E2 -25387.135} C_VEL
LIN {X 0,Y 122.36,Z 635.216,A -85,B 0,C 180,E1 -25392.471,E2 -25392.471} C_VEL
LIN {X 0,Y 122.041,Z 635.279,A -85,B 0,C 180,E1 -25400.212,E2 -25400.212} C_VEL
LIN {X 0,Y 121.979,Z 635.268,A -85,B 0,C 180,E1 -25403.784,E2 -25403.784} C_VEL
LIN {X 0,Y 121.925,Z 635.292,A -85,B 0,C 180,E1 -25410.162,E2 -25410.162} C_VEL
LIN {X 0,Y 121.932,Z 635.277,A -85,B 0,C 180,E1 -25416.204,E2 -25416.204} C_VEL
LIN {X 0,Y 121.938,Z 635.29,A -85,B 0,C 180,E1 -25421.475,E2 -25421.475} C_VEL
LIN {X 0,Y 121.926,Z 635.277,A -85,B 0,C 180,E1 -25428.53,E2 -25428.53} C_VEL
LIN {X 0,Y 121.943,Z 635.296,A -85,B 0,C 180,E1 -25434.808,E2 -25434.808} C_VEL
LIN {X 0,Y 121.926,Z 635.281,A -85,B 0,C 180,E1 -25439.836,E2 -25439.836} C_VEL
LIN {X 0,Y 121.98,Z 635.288,A -85,B 0,C 180,E1 -25446.215,E2 -25446.215} C_VEL
LIN {X 0,Y 122.048,Z 635.279,A -85,B 0,C 180,E1 -25449.788,E2 -25449.788} C_VEL
LIN {X 0,Y 122.262,Z 635.251,A -85,B 0,C 180,E1 -25456.707,E2 -25456.707} C_VEL
LIN {X 0,Y 122.438,Z 635.228,A -85,B 0,C 180,E1 -25461.438,E2 -25461.438} C_VEL
LIN {X 0,Y 123.45,Z 638.087,A -85,B 0,C 180,E1 -25462.09,E2 -25462.09} C_VEL
LIN {X 0,Y 125.223,Z 640.575,A -85,B 0,C 180,E1 -25462.963,E2 -25462.963} C_VEL
LIN {X 0,Y 132.247,Z 651.96,A -85,B 0,C 180,E1 -25466.313,E2 -25466.313} C_VEL
LIN {X 0,Y 141.084,Z 670.76,A -85,B 0,C 180,E1 -25470.262,E2 -25470.262} C_VEL
LIN {X 0,Y 146.268,Z 683.321,A -85,B 0,C 180,E1 -25472.439,E2 -25472.439} C_VEL
LIN {X 0,Y 142.501,Z 729.981,A -85,B 0,C 180,E1 -25474.959,E2 -25474.959} C_VEL
LIN {X 0,Y 140.751,Z 743.931,A -85,B 0,C 180,E1 -25476.269,E2 -25476.269} C_VEL
LIN {X 0,Y 138.449,Z 756.723,A -85,B 0,C 180,E1 -25478.024,E2 -25478.024} C_VEL
LIN {X 0,Y 135.737,Z 769.016,A -85,B 0,C 180,E1 -25480.35,E2 -25480.35} C_VEL
LIN {X 0,Y 132.777,Z 779.85,A -85,B 0,C 180,E1 -25483,E2 -25483} C_VEL
LIN {X 0,Y 129.608,Z 790.834,A -85,B 0,C 180,E1 -25486.539,E2 -25486.539} C_VEL
LIN {X 0,Y 126.55,Z 800.45,A -85,B 0,C 180,E1 -25490.516,E2 -25490.516} C_VEL
LIN {X 0,Y 123.934,Z 808.681,A -85,B 0,C 180,E1 -25494.867,E2 -25494.867} C_VEL
LIN {X 0,Y 121.716,Z 816.165,A -85,B 0,C 180,E1 -25499.994,E2 -25499.994} C_VEL
LIN {X 0,Y 120.24,Z 821.921,A -85,B 0,C 180,E1 -25505.089,E2 -25505.089} C_VEL
LIN {X 0,Y 119.256,Z 826.527,A -85,B 0,C 180,E1 -25510.409,E2 -25510.409} C_VEL
LIN {X 0,Y 118.981,Z 829.594,A -85,B 0,C 180,E1 -25515.137,E2 -25515.137} C_VEL
LIN {X 0,Y 119.404,Z 831.856,A -85,B 0,C 180,E1 -25519.92,E2 -25519.92} C_VEL
LIN {X 0,Y 120.53,Z 833.335,A -85,B 0,C 180,E1 -25524.717,E2 -25524.717} C_VEL
LIN {X 0,Y 122.301,Z 833.995,A -85,B 0,C 180,E1 -25529.536,E2 -25529.536} C_VEL
LIN {X 0,Y 124.867,Z 833.816,A -85,B 0,C 180,E1 -25534.226,E2 -25534.226} C_VEL
LIN {X 0,Y 128.19,Z 832.804,A -85,B 0,C 180,E1 -25538.749,E2 -25538.749} C_VEL
LIN {X 0,Y 132.237,Z 830.922,A -85,B 0,C 180,E1 -25543.062,E2 -25543.062} C_VEL
LIN {X 0,Y 138.587,Z 827.049,A -85,B 0,C 180,E1 -25548.298,E2 -25548.298} C_VEL
LIN {X 0,Y 144.77,Z 822.481,A -85,B 0,C 180,E1 -25552.316,E2 -25552.316} C_VEL
LIN {X 0,Y 151.673,Z 816.44,A -85,B 0,C 180,E1 -25556.016,E2 -25556.016} C_VEL
LIN {X 0,Y 157.709,Z 810.352,A -85,B 0,C 180,E1 -25558.765,E2 -25558.765} C_VEL
LIN {X 0,Y 165.724,Z 800.913,A -85,B 0,C 180,E1 -25561.914,E2 -25561.914} C_VEL
LIN {X 0,Y 171.403,Z 793.124,A -85,B 0,C 180,E1 -25563.852,E2 -25563.852} C_VEL
LIN {X 0,Y 177.419,Z 783.56,A -85,B 0,C 180,E1 -25565.682,E2 -25565.682} C_VEL
LIN {X 0,Y 183.099,Z 772.556,A -85,B 0,C 180,E1 -25567.313,E2 -25567.313} C_VEL
LIN {X 0,Y 188.365,Z 759.887,A -85,B 0,C 180,E1 -25568.711,E2 -25568.711} C_VEL
LIN {X 0,Y 192.216,Z 747.54,A -85,B 0,C 180,E1 -25569.748,E2 -25569.748} C_VEL
LIN {X 0,Y 195.242,Z 734.317,A -85,B 0,C 180,E1 -25570.461,E2 -25570.461} C_VEL
LIN {X 0,Y 197.457,Z 718.964,A -85,B 0,C 180,E1 -25571.047,E2 -25571.047} C_VEL
LIN {X 0,Y 195.661,Z 714.949,A -85,B 0,C 180,E1 -25574.119,E2 -25574.119} C_VEL
LIN {X 0,Y 194.794,Z 712.914,A -85,B 0,C 180,E1 -25576.3,E2 -25576.3} C_VEL
LIN {X 0,Y 193.944,Z 711.334,A -85,B 0,C 180,E1 -25579.585,E2 -25579.585} C_VEL
LIN {X 0,Y 193.694,Z 711.799,A -85,B 0,C 180,E1 -25583.525,E2 -25583.525} C_VEL
LIN {X 0,Y 194.055,Z 714.522,A -85,B 0,C 180,E1 -25586.824,E2 -25586.824} C_VEL
LIN {X 0,Y 194.741,Z 716.92,A -85,B 0,C 180,E1 -25589.081,E2 -25589.081} C_VEL
LIN {X 0,Y 195.711,Z 720.768,A -85,B 0,C 180,E1 -25591.46,E2 -25591.46} C_VEL
LIN {X 0,Y 196.795,Z 725.263,A -85,B 0,C 180,E1 -25593.595,E2 -25593.595} C_VEL
LIN {X 0,Y 194.095,Z 742.477,A -85,B 0,C 180,E1 -25594.228,E2 -25594.228} C_VEL
LIN {X 0,Y 190.902,Z 755.11,A -85,B 0,C 180,E1 -25594.869,E2 -25594.869} C_VEL
LIN {X 0,Y 186.327,Z 768.25,A -85,B 0,C 180,E1 -25595.813,E2 -25595.813} C_VEL
LIN {X 0,Y 181.3,Z 779.562,A -85,B 0,C 180,E1 -25596.918,E2 -25596.918} C_VEL
LIN {X 0,Y 175.066,Z 791.03,A -85,B 0,C 180,E1 -25598.482,E2 -25598.482} C_VEL
LIN {X 0,Y 168.377,Z 801.347,A -85,B 0,C 180,E1 -25600.383,E2 -25600.383} C_VEL
LIN {X 0,Y 160.656,Z 811.416,A -85,B 0,C 180,E1 -25602.885,E2 -25602.885} C_VEL
LIN {X 0,Y 153.526,Z 819.557,A -85,B 0,C 180,E1 -25605.726,E2 -25605.726} C_VEL
LIN {X 0,Y 146.898,Z 826.209,A -85,B 0,C 180,E1 -25608.866,E2 -25608.866} C_VEL
LIN {X 0,Y 139.794,Z 832.434,A -85,B 0,C 180,E1 -25612.895,E2 -25612.895} C_VEL
LIN {X 0,Y 134.637,Z 836.498,A -85,B 0,C 180,E1 -25616.639,E2 -25616.639} C_VEL
LIN {X 0,Y 129.901,Z 839.779,A -85,B 0,C 180,E1 -25620.862,E2 -25620.862} C_VEL
LIN {X 0,Y 124.929,Z 842.67,A -85,B 0,C 180,E1 -25626.81,E2 -25626.81} C_VEL
LIN {X 0,Y 121.528,Z 844.016,A -85,B 0,C 180,E1 -25633.193,E2 -25633.193} C_VEL
LIN {X 0,Y 119.856,Z 843.919,A -85,B 0,C 180,E1 -25639.869,E2 -25639.869} C_VEL
LIN {X 0,Y 119.585,Z 843.307,A -85,B 0,C 180,E1 -25643.25,E2 -25643.25} C_VEL
LIN {X 0,Y 119.673,Z 842.241,A -85,B 0,C 180,E1 -25646.741,E2 -25646.741} C_VEL
LIN {X 0,Y 119.931,Z 840.849,A -85,B 0,C 180,E1 -25650,E2 -25650} C_VEL
LIN {X 0,Y 119.729,Z 837.737,A -85,B 0,C 180,E1 -25655.05,E2 -25655.05} C_VEL
LIN {X 0,Y 120.074,Z 833.475,A -85,B 0,C 180,E1 -25660.113,E2 -25660.113} C_VEL
LIN {X 0,Y 121.082,Z 827.95,A -85,B 0,C 180,E1 -25665.141,E2 -25665.141} C_VEL
LIN {X 0,Y 122.985,Z 821.015,A -85,B 0,C 180,E1 -25670.051,E2 -25670.051} C_VEL
LIN {X 0,Y 123.876,Z 817.962,A -85,B 0,C 180,E1 -25671.852,E2 -25671.852} C_VEL
LIN {X 0,Y 124.34,Z 814.162,A -85,B 0,C 180,E1 -25673.94,E2 -25673.94} C_VEL
LIN {X 0,Y 123.517,Z 807.47,A -85,B 0,C 180,E1 -25677.329,E2 -25677.329} C_VEL
LIN {X 0,Y 123.028,Z 800.24,A -85,B 0,C 180,E1 -25680.493,E2 -25680.493} C_VEL
LIN {X 0,Y 123.974,Z 795.597,A -85,B 0,C 180,E1 -25682.136,E2 -25682.136} C_VEL
LIN {X 0,Y 127.462,Z 784.095,A -85,B 0,C 180,E1 -25685.375,E2 -25685.375} C_VEL
LIN {X 0,Y 130.499,Z 772.757,A -85,B 0,C 180,E1 -25687.776,E2 -25687.776} C_VEL
LIN {X 0,Y 133.245,Z 760.009,A -85,B 0,C 180,E1 -25689.756,E2 -25689.756} C_VEL
LIN {X 0,Y 135.367,Z 746.807,A -85,B 0,C 180,E1 -25691.2,E2 -25691.2} C_VEL
LIN {X 0,Y 136.906,Z 731.696,A -85,B 0,C 180,E1 -25692.204,E2 -25692.204} C_VEL
LIN {X 0,Y 139.136,Z 702.309,A -85,B 0,C 180,E1 -25693.853,E2 -25693.853} C_VEL
LIN {X 0,Y 138.041,Z 689.247,A -85,B 0,C 180,E1 -25695.103,E2 -25695.103} C_VEL
LIN {X 0,Y 132.487,Z 672.578,A -85,B 0,C 180,E1 -25697.921,E2 -25697.921} C_VEL
LIN {X 0,Y 126.505,Z 657.453,A -85,B 0,C 180,E1 -25701.055,E2 -25701.055} C_VEL
LIN {X 0,Y 122.834,Z 649.909,A -85,B 0,C 180,E1 -25703.037,E2 -25703.037} C_VEL
LIN {X 0,Y 119.098,Z 643.912,A -85,B 0,C 180,E1 -25705.003,E2 -25705.003} C_VEL
LIN {X 0,Y 117.097,Z 640.535,A -85,B 0,C 180,E1 -25706.146,E2 -25706.146} C_VEL
LIN {X 0,Y 115.33,Z 638.024,A -85,B 0,C 180,E1 -25707.157,E2 -25707.157} C_VEL
LIN {X 0,Y 114.824,Z 636.181,A -85,B 0,C 180,E1 -25707.582,E2 -25707.582} C_VEL
LIN {X 0,Y 114.859,Z 636.177,A -85,B 0,C 180,E1 -25710.69,E2 -25710.69} C_VEL
LIN {X 0,Y 114.946,Z 636.166,A -85,B 0,C 180,E1 -25716.506,E2 -25716.506} C_VEL
LIN {X 0,Y 115.001,Z 636.148,A -85,B 0,C 180,E1 -25722.206,E2 -25722.206} C_VEL
LIN {X 0,Y 115.282,Z 636.123,A -85,B 0,C 180,E1 -25727.262,E2 -25727.262} C_VEL
LIN {X 0,Y 115.383,Z 636.106,A -85,B 0,C 180,E1 -25733.001,E2 -25733.001} C_VEL
LIN {X 0,Y 115.992,Z 636.015,A -85,B 0,C 180,E1 -25739.998,E2 -25739.998} C_VEL
LIN {X 0,Y 115.383,Z 636.111,A -85,B 0,C 180,E1 -25747.024,E2 -25747.024} C_VEL
LIN {X 0,Y 115.281,Z 636.096,A -85,B 0,C 180,E1 -25752.735,E2 -25752.735} C_VEL
LIN {X 0,Y 115.008,Z 636.154,A -85,B 0,C 180,E1 -25757.789,E2 -25757.789} C_VEL
LIN {X 0,Y 114.943,Z 636.146,A -85,B 0,C 180,E1 -25763.491,E2 -25763.491} C_VEL
LIN {X 0,Y 114.86,Z 636.174,A -85,B 0,C 180,E1 -25771.063,E2 -25771.063} C_VEL
LIN {X 0,Y 114.844,Z 636.152,A -85,B 0,C 180,E1 -25777.729,E2 -25777.729} C_VEL
LIN {X 0,Y 114.861,Z 636.176,A -85,B 0,C 180,E1 -25782.758,E2 -25782.758} C_VEL
LIN {X 0,Y 114.856,Z 636.162,A -85,B 0,C 180,E1 -25787.696,E2 -25787.696} C_VEL
LIN {X 0,Y 114.82,Z 636.177,A -85,B 0,C 180,E1 -25792.719,E2 -25792.719} C_VEL
LIN {X 0,Y 114.86,Z 636.16,A -85,B 0,C 180,E1 -25798.936,E2 -25798.936} C_VEL
LIN {X 0,Y 114.945,Z 636.165,A -85,B 0,C 180,E1 -25806.506,E2 -25806.506} C_VEL
LIN {X 0,Y 115.017,Z 636.155,A -85,B 0,C 180,E1 -25812.211,E2 -25812.211} C_VEL
LIN {X 0,Y 115.329,Z 636.114,A -85,B 0,C 180,E1 -25818.561,E2 -25818.561} C_VEL
LIN {X 0,Y 116.439,Z 639.093,A -85,B 0,C 180,E1 -25819.403,E2 -25819.403} C_VEL
LIN {X 0,Y 118.083,Z 641.219,A -85,B 0,C 180,E1 -25820.306,E2 -25820.306} C_VEL
LIN {X 0,Y 127.163,Z 655.907,A -85,B 0,C 180,E1 -25825.006,E2 -25825.006} C_VEL
LIN {X 0,Y 135.928,Z 675.01,A -85,B 0,C 180,E1 -25829.214,E2 -25829.214} C_VEL
LIN {X 0,Y 140.021,Z 685.112,A -85,B 0,C 180,E1 -25831.056,E2 -25831.056} C_VEL
LIN {X 0,Y 136.224,Z 730.356,A -85,B 0,C 180,E1 -25833.586,E2 -25833.586} C_VEL
LIN {X 0,Y 134.369,Z 744.596,A -85,B 0,C 180,E1 -25834.98,E2 -25834.98} C_VEL
LIN {X 0,Y 132.115,Z 756.625,A -85,B 0,C 180,E1 -25836.682,E2 -25836.682} C_VEL
LIN {X 0,Y 129.383,Z 768.508,A -85,B 0,C 180,E1 -25838.984,E2 -25838.984} C_VEL
LIN {X 0,Y 126.303,Z 779.37,A -85,B 0,C 180,E1 -25841.711,E2 -25841.711} C_VEL
LIN {X 0,Y 123.299,Z 789.455,A -85,B 0,C 180,E1 -25844.996,E2 -25844.996} C_VEL
LIN {X 0,Y 119.961,Z 799.636,A -85,B 0,C 180,E1 -25849.295,E2 -25849.295} C_VEL
LIN {X 0,Y 117.146,Z 808.087,A -85,B 0,C 180,E1 -25853.888,E2 -25853.888} C_VEL
LIN {X 0,Y 114.768,Z 815.821,A -85,B 0,C 180,E1 -25859.333,E2 -25859.333} C_VEL
LIN {X 0,Y 113.384,Z 820.933,A -85,B 0,C 180,E1 -25863.907,E2 -25863.907} C_VEL
LIN {X 0,Y 112.379,Z 825.204,A -85,B 0,C 180,E1 -25868.709,E2 -25868.709} C_VEL
LIN {X 0,Y 111.913,Z 828.65,A -85,B 0,C 180,E1 -25873.691,E2 -25873.691} C_VEL
LIN {X 0,Y 112.151,Z 831.283,A -85,B 0,C 180,E1 -25878.761,E2 -25878.761} C_VEL
LIN {X 0,Y 113.826,Z 833.718,A -85,B 0,C 180,E1 -25886.244,E2 -25886.244} C_VEL
LIN {X 0,Y 115.679,Z 834.346,A -85,B 0,C 180,E1 -25890.922,E2 -25890.922} C_VEL
LIN {X 0,Y 118.234,Z 834.291,A -85,B 0,C 180,E1 -25895.414,E2 -25895.414} C_VEL
LIN {X 0,Y 121.405,Z 833.576,A -85,B 0,C 180,E1 -25899.678,E2 -25899.678} C_VEL
LIN {X 0,Y 127.232,Z 831.172,A -85,B 0,C 180,E1 -25905.609,E2 -25905.609} C_VEL
LIN {X 0,Y 134.257,Z 827.214,A -85,B 0,C 180,E1 -25910.966,E2 -25910.966} C_VEL
LIN {X 0,Y 141.079,Z 822.413,A -85,B 0,C 180,E1 -25915.067,E2 -25915.067} C_VEL
LIN {X 0,Y 149.514,Z 815.31,A -85,B 0,C 180,E1 -25919.171,E2 -25919.171} C_VEL
LIN {X 0,Y 156.343,Z 808.592,A -85,B 0,C 180,E1 -25921.924,E2 -25921.924} C_VEL
LIN {X 0,Y 163.757,Z 799.983,A -85,B 0,C 180,E1 -25924.578,E2 -25924.578} C_VEL
LIN {X 0,Y 170.541,Z 790.716,A -85,B 0,C 180,E1 -25926.659,E2 -25926.659} C_VEL
LIN {X 0,Y 177.017,Z 780.212,A -85,B 0,C 180,E1 -25928.451,E2 -25928.451} C_VEL
LIN {X 0,Y 182.415,Z 769.598,A -85,B 0,C 180,E1 -25929.846,E2 -25929.846} C_VEL
LIN {X 0,Y 187.296,Z 757.488,A -85,B 0,C 180,E1 -25931.05,E2 -25931.05} C_VEL
LIN {X 0,Y 190.78,Z 746.249,A -85,B 0,C 180,E1 -25931.895,E2 -25931.895} C_VEL
LIN {X 0,Y 193.673,Z 733.468,A -85,B 0,C 180,E1 -25932.529,E2 -25932.529} C_VEL
LIN {X 0,Y 195.086,Z 723.922,A -85,B 0,C 180,E1 -25932.891,E2 -25932.891} C_VEL
LIN {X 0,Y 194.157,Z 721.434,A -85,B 0,C 180,E1 -25934.88,E2 -25934.88} C_VEL
LIN {X 0,Y 193.518,Z 719.808,A -85,B 0,C 180,E1 -25936.644,E2 -25936.644} C_VEL
LIN {X 0,Y 192.755,Z 718.326,A -85,B 0,C 180,E1 -25939.938,E2 -25939.938} C_VEL
LIN {X 0,Y 192.553,Z 718.84,A -85,B 0,C 180,E1 -25943.447,E2 -25943.447} C_VEL
LIN {X 0,Y 193.243,Z 722.929,A -85,B 0,C 180,E1 -25948.058,E2 -25948.058} C_VEL
LIN {X 0,Y 194.08,Z 727.16,A -85,B 0,C 180,E1 -25950.689,E2 -25950.689} C_VEL
LIN {X 0,Y 194.514,Z 729.397,A -85,B 0,C 180,E1 -25951.738,E2 -25951.738} C_VEL
LIN {X 0,Y 192.001,Z 743.613,A -85,B 0,C 180,E1 -25952.239,E2 -25952.239} C_VEL
LIN {X 0,Y 188.106,Z 757.584,A -85,B 0,C 180,E1 -25952.957,E2 -25952.957} C_VEL
LIN {X 0,Y 183.864,Z 768.892,A -85,B 0,C 180,E1 -25953.762,E2 -25953.762} C_VEL
LIN {X 0,Y 177.961,Z 781.245,A -85,B 0,C 180,E1 -25954.972,E2 -25954.972} C_VEL
LIN {X 0,Y 171.534,Z 792.329,A -85,B 0,C 180,E1 -25956.482,E2 -25956.482} C_VEL
LIN {X 0,Y 165.329,Z 801.428,A -85,B 0,C 180,E1 -25958.149,E2 -25958.149} C_VEL
LIN {X 0,Y 158.63,Z 809.875,A -85,B 0,C 180,E1 -25960.161,E2 -25960.161} C_VEL
LIN {X 0,Y 151.019,Z 818.195,A -85,B 0,C 180,E1 -25962.866,E2 -25962.866} C_VEL
LIN {X 0,Y 143.91,Z 824.99,A -85,B 0,C 180,E1 -25965.901,E2 -25965.901} C_VEL
LIN {X 0,Y 136.253,Z 831.378,A -85,B 0,C 180,E1 -25969.854,E2 -25969.854} C_VEL
LIN {X 0,Y 130.445,Z 835.657,A -85,B 0,C 180,E1 -25973.656,E2 -25973.656} C_VEL
LIN {X 0,Y 123.751,Z 839.894,A -85,B 0,C 180,E1 -25979.262,E2 -25979.262} C_VEL
LIN {X 0,Y 118.423,Z 842.53,A -85,B 0,C 180,E1 -25985.454,E2 -25985.454} C_VEL
LIN {X 0,Y 114.707,Z 843.704,A -85,B 0,C 180,E1 -25992.161,E2 -25992.161} C_VEL
LIN {X 0,Y 112.852,Z 843.406,A -85,B 0,C 180,E1 -25999.233,E2 -25999.233} C_VEL
LIN {X 0,Y 112.603,Z 841.573,A -85,B 0,C 180,E1 -26006.422,E2 -26006.422} C_VEL
LIN {X 0,Y 112.87,Z 840.059,A -85,B 0,C 180,E1 -26010,E2 -26010} C_VEL
LIN {X 0,Y 112.672,Z 836.778,A -85,B 0,C 180,E1 -26015.368,E2 -26015.368} C_VEL
LIN {X 0,Y 113.084,Z 832.351,A -85,B 0,C 180,E1 -26020.745,E2 -26020.745} C_VEL
LIN {X 0,Y 114.233,Z 826.65,A -85,B 0,C 180,E1 -26026.072,E2 -26026.072} C_VEL
LIN {X 0,Y 116.322,Z 819.452,A -85,B 0,C 180,E1 -26031.254,E2 -26031.254} C_VEL
LIN {X 0,Y 119.103,Z 810.411,A -85,B 0,C 180,E1 -26036.267,E2 -26036.267} C_VEL
LIN {X 0,Y 122.375,Z 800.662,A -85,B 0,C 180,E1 -26040.385,E2 -26040.385} C_VEL
LIN {X 0,Y 123.974,Z 795.597,A -85,B 0,C 180,E1 -26042.136,E2 -26042.136} C_VEL
LIN {X 0,Y 124.924,Z 790.907,A -85,B 0,C 180,E1 -26043.653,E2 -26043.653} C_VEL
LIN {X 0,Y 124.626,Z 782.858,A -85,B 0,C 180,E1 -26046.244,E2 -26046.244} C_VEL
LIN {X 0,Y 124.183,Z 774.277,A -85,B 0,C 180,E1 -26048.637,E2 -26048.637} C_VEL
LIN {X 0,Y 124.907,Z 768.802,A -85,B 0,C 180,E1 -26049.785,E2 -26049.785} C_VEL
LIN {X 0,Y 127.373,Z 757.569,A -85,B 0,C 180,E1 -26051.46,E2 -26051.46} C_VEL
LIN {X 0,Y 129.453,Z 744.129,A -85,B 0,C 180,E1 -26052.867,E2 -26052.867} C_VEL
LIN {X 0,Y 131.317,Z 724.865,A -85,B 0,C 180,E1 -26054.086,E2 -26054.086} C_VEL
LIN {X 0,Y 133.05,Z 703.271,A -85,B 0,C 180,E1 -26055.336,E2 -26055.336} C_VEL
LIN {X 0,Y 132.118,Z 691.509,A -85,B 0,C 180,E1 -26056.51,E2 -26056.51} C_VEL
LIN {X 0,Y 126.985,Z 675.819,A -85,B 0,C 180,E1 -26059.303,E2 -26059.303} C_VEL
LIN {X 0,Y 121.493,Z 661.434,A -85,B 0,C 180,E1 -26062.466,E2 -26062.466} C_VEL
LIN {X 0,Y 117.665,Z 653.508,A -85,B 0,C 180,E1 -26064.644,E2 -26064.644} C_VEL
LIN {X 0,Y 112.519,Z 645.277,A -85,B 0,C 180,E1 -26067.665,E2 -26067.665} C_VEL
LIN {X 0,Y 110.041,Z 641.364,A -85,B 0,C 180,E1 -26069.272,E2 -26069.272} C_VEL
LIN {X 0,Y 108.39,Z 639.111,A -85,B 0,C 180,E1 -26070.367,E2 -26070.367} C_VEL
LIN {X 0,Y 107.813,Z 637.055,A -85,B 0,C 180,E1 -26070.997,E2 -26070.997} C_VEL
LIN {X 0,Y 107.909,Z 637.044,A -85,B 0,C 180,E1 -26076.995,E2 -26076.995} C_VEL
LIN {X 0,Y 108.031,Z 637.029,A -85,B 0,C 180,E1 -26084.915,E2 -26084.915} C_VEL
LIN {X 0,Y 108.285,Z 636.984,A -85,B 0,C 180,E1 -26088.77,E2 -26088.77} C_VEL
LIN {X 0,Y 108.453,Z 636.975,A -85,B 0,C 180,E1 -26096.283,E2 -26096.283} C_VEL
LIN {X 0,Y 108.918,Z 636.895,A -85,B 0,C 180,E1 -26099.998,E2 -26099.998} C_VEL
LIN {X 0,Y 108.325,Z 636.991,A -85,B 0,C 180,E1 -26107.454,E2 -26107.454} C_VEL
LIN {X 0,Y 108.196,Z 636.977,A -85,B 0,C 180,E1 -26113.013,E2 -26113.013} C_VEL
LIN {X 0,Y 107.901,Z 637.041,A -85,B 0,C 180,E1 -26119.004,E2 -26119.004} C_VEL
LIN {X 0,Y 107.852,Z 637.023,A -85,B 0,C 180,E1 -26124.18,E2 -26124.18} C_VEL
LIN {X 0,Y 107.792,Z 637.057,A -85,B 0,C 180,E1 -26132.051,E2 -26132.051} C_VEL
LIN {X 0,Y 107.75,Z 637.035,A -85,B 0,C 180,E1 -26138.494,E2 -26138.494} C_VEL
LIN {X 0,Y 107.76,Z 637.057,A -85,B 0,C 180,E1 -26145.838,E2 -26145.838} C_VEL
LIN {X 0,Y 107.725,Z 637.051,A -85,B 0,C 180,E1 -26151.522,E2 -26151.522} C_VEL
LIN {X 0,Y 107.799,Z 637.04,A -85,B 0,C 180,E1 -26158.564,E2 -26158.564} C_VEL
LIN {X 0,Y 107.909,Z 637.043,A -85,B 0,C 180,E1 -26166.998,E2 -26166.998} C_VEL
LIN {X 0,Y 108.06,Z 637.021,A -85,B 0,C 180,E1 -26175.167,E2 -26175.167} C_VEL
LIN {X 0,Y 109.215,Z 639.995,A -85,B 0,C 180,E1 -26176.143,E2 -26176.143} C_VEL
LIN {X 0,Y 111.345,Z 642.48,A -85,B 0,C 180,E1 -26177.442,E2 -26177.442} C_VEL
LIN {X 0,Y 114.41,Z 647.484,A -85,B 0,C 180,E1 -26179.381,E2 -26179.381} C_VEL
LIN {X 0,Y 121.567,Z 658.978,A -85,B 0,C 180,E1 -26183.336,E2 -26183.336} C_VEL
LIN {X 0,Y 130.051,Z 677.432,A -85,B 0,C 180,E1 -26187.747,E2 -26187.747} C_VEL
LIN {X 0,Y 133.842,Z 687.391,A -85,B 0,C 180,E1 -26189.619,E2 -26189.619} C_VEL
LIN {X 0,Y 129.976,Z 730.794,A -85,B 0,C 180,E1 -26192.13,E2 -26192.13} C_VEL
LIN {X 0,Y 128.092,Z 744.686,A -85,B 0,C 180,E1 -26193.54,E2 -26193.54} C_VEL
LIN {X 0,Y 125.649,Z 757.069,A -85,B 0,C 180,E1 -26195.353,E2 -26195.353} C_VEL
LIN {X 0,Y 122.75,Z 769.186,A -85,B 0,C 180,E1 -26197.815,E2 -26197.815} C_VEL
LIN {X 0,Y 119.621,Z 779.715,A -85,B 0,C 180,E1 -26200.579,E2 -26200.579} C_VEL
LIN {X 0,Y 116.524,Z 789.641,A -85,B 0,C 180,E1 -26203.96,E2 -26203.96} C_VEL
LIN {X 0,Y 113.32,Z 799.029,A -85,B 0,C 180,E1 -26208.065,E2 -26208.065} C_VEL
LIN {X 0,Y 110.574,Z 806.872,A -85,B 0,C 180,E1 -26212.417,E2 -26212.417} C_VEL
LIN {X 0,Y 108.03,Z 814.781,A -85,B 0,C 180,E1 -26218.046,E2 -26218.046} C_VEL
LIN {X 0,Y 106.482,Z 820.217,A -85,B 0,C 180,E1 -26222.991,E2 -26222.991} C_VEL
LIN {X 0,Y 105.157,Z 825.7,A -85,B 0,C 180,E1 -26229.41,E2 -26229.41} C_VEL
LIN {X 0,Y 104.8,Z 829.167,A -85,B 0,C 180,E1 -26234.852,E2 -26234.852} C_VEL
LIN {X 0,Y 104.964,Z 830.763,A -85,B 0,C 180,E1 -26237.969,E2 -26237.969} C_VEL
LIN {X 0,Y 105.815,Z 832.85,A -85,B 0,C 180,E1 -26243.293,E2 -26243.293} C_VEL
LIN {X 0,Y 107.383,Z 834.173,A -85,B 0,C 180,E1 -26248.429,E2 -26248.429} C_VEL
LIN {X 0,Y 109.791,Z 834.789,A -85,B 0,C 180,E1 -26253.656,E2 -26253.656} C_VEL
LIN {X 0,Y 113.107,Z 834.566,A -85,B 0,C 180,E1 -26258.752,E2 -26258.752} C_VEL
LIN {X 0,Y 117.232,Z 833.521,A -85,B 0,C 180,E1 -26263.57,E2 -26263.57} C_VEL
LIN {X 0,Y 122.117,Z 831.622,A -85,B 0,C 180,E1 -26268.056,E2 -26268.056} C_VEL
LIN {X 0,Y 127.692,Z 828.825,A -85,B 0,C 180,E1 -26272.169,E2 -26272.169} C_VEL
LIN {X 0,Y 135.989,Z 823.648,A -85,B 0,C 180,E1 -26277.039,E2 -26277.039} C_VEL
LIN {X 0,Y 143.7,Z 817.821,A -85,B 0,C 180,E1 -26280.662,E2 -26280.662} C_VEL
LIN {X 0,Y 152.174,Z 810.117,A -85,B 0,C 180,E1 -26283.975,E2 -26283.975} C_VEL
LIN {X 0,Y 160.015,Z 801.671,A -85,B 0,C 180,E1 -26286.622,E2 -26286.622} C_VEL
LIN {X 0,Y 166.65,Z 793.325,A -85,B 0,C 180,E1 -26288.548,E2 -26288.548} C_VEL
LIN {X 0,Y 174.037,Z 782.132,A -85,B 0,C 180,E1 -26290.471,E2 -26290.471} C_VEL
LIN {X 0,Y 179.821,Z 771.426,A -85,B 0,C 180,E1 -26291.861,E2 -26291.861} C_VEL
LIN {X 0,Y 185.014,Z 759.356,A -85,B 0,C 180,E1 -26293.051,E2 -26293.051} C_VEL
LIN {X 0,Y 189.022,Z 747.164,A -85,B 0,C 180,E1 -26293.953,E2 -26293.953} C_VEL
LIN {X 0,Y 192.046,Z 734.516,A -85,B 0,C 180,E1 -26294.56,E2 -26294.56} C_VEL
LIN {X 0,Y 193.018,Z 728.798,A -85,B 0,C 180,E1 -26294.767,E2 -26294.767} C_VEL
LIN {X 0,Y 192.246,Z 726.679,A -85,B 0,C 180,E1 -26297.006,E2 -26297.006} C_VEL
LIN {X 0,Y 191.715,Z 725.607,A -85,B 0,C 180,E1 -26299.265,E2 -26299.265} C_VEL
LIN {X 0,Y 191.383,Z 725.568,A -85,B 0,C 180,E1 -26302.428,E2 -26302.428} C_VEL
LIN {X 0,Y 191.408,Z 726.493,A -85,B 0,C 180,E1 -26304.071,E2 -26304.071} C_VEL
LIN {X 0,Y 191.922,Z 730.044,A -85,B 0,C 180,E1 -26307.696,E2 -26307.696} C_VEL
LIN {X 0,Y 192.422,Z 733.351,A -85,B 0,C 180,E1 -26309.778,E2 -26309.778} C_VEL
LIN {X 0,Y 189.398,Z 747.686,A -85,B 0,C 180,E1 -26310.345,E2 -26310.345} C_VEL
LIN {X 0,Y 185.558,Z 759.887,A -85,B 0,C 180,E1 -26310.976,E2 -26310.976} C_VEL
LIN {X 0,Y 180.155,Z 772.928,A -85,B 0,C 180,E1 -26311.955,E2 -26311.955} C_VEL
LIN {X 0,Y 174.119,Z 784.408,A -85,B 0,C 180,E1 -26313.121,E2 -26313.121} C_VEL
LIN {X 0,Y 166.801,Z 795.787,A -85,B 0,C 180,E1 -26314.755,E2 -26314.755} C_VEL
LIN {X 0,Y 159.735,Z 805.055,A -85,B 0,C 180,E1 -26316.588,E2 -26316.588} C_VEL
LIN {X 0,Y 151.505,Z 814.232,A -85,B 0,C 180,E1 -26319.016,E2 -26319.016} C_VEL
LIN {X 0,Y 142.535,Z 822.781,A -85,B 0,C 180,E1 -26322.303,E2 -26322.303} C_VEL
LIN {X 0,Y 135.412,Z 828.65,A -85,B 0,C 180,E1 -26325.521,E2 -26325.521} C_VEL
LIN {X 0,Y 128.799,Z 833.391,A -85,B 0,C 180,E1 -26329.098,E2 -26329.098} C_VEL
LIN {X 0,Y 122.263,Z 837.522,A -85,B 0,C 180,E1 -26333.589,E2 -26333.589} C_VEL
LIN {X 0,Y 117.691,Z 839.966,A -85,B 0,C 180,E1 -26337.491,E2 -26337.491} C_VEL
LIN {X 0,Y 111.994,Z 842.396,A -85,B 0,C 180,E1 -26343.943,E2 -26343.943} C_VEL
LIN {X 0,Y 109.705,Z 843.071,A -85,B 0,C 180,E1 -26347.395,E2 -26347.395} C_VEL
LIN {X 0,Y 106.707,Z 843.28,A -85,B 0,C 180,E1 -26354.725,E2 -26354.725} C_VEL
